Yaskawa INFORM job: DEMO_ROOF_SIDE_0625_3PAINT_11.JBI

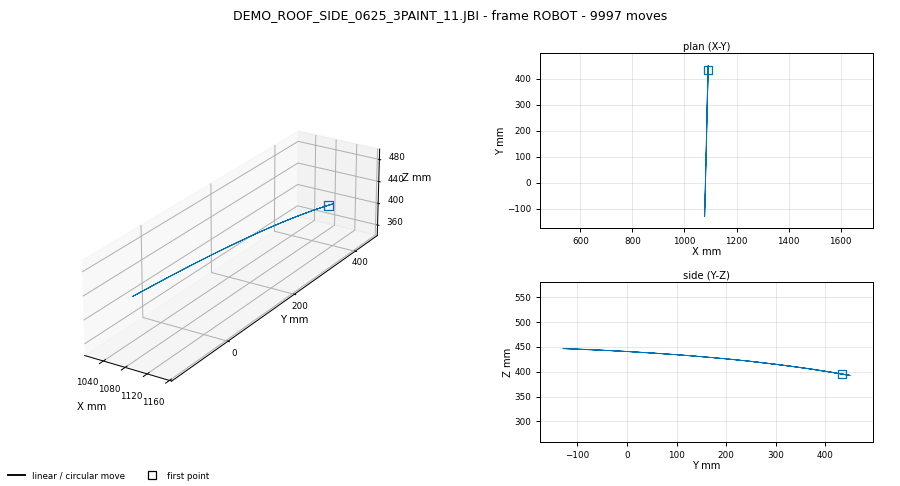
[picture p0: tool path of DEMO_ROOF_SIDE_0625_3PAINT_11.JBI in frame ROBOT, 9997 of 9997 moves have a stored position in this frame; points joined in program order, loops and branches not executed]
/JOB
//NAME DEMO_ROOF_SIDE_0625_3PAINT11
//POS
///NPOS 9997,0,0,0,0,0
///TOOL 0
///USER 0
///POSTYPE ROBOT
///RECTAN
///RCONF 1,0,0,0,0,0,0,0,0,0,0,0,0,0,0,0,0,0,0,0,0,0,0,0
C00000=1091.874,433.807,395.895,178.473,26.068,154.099
C00001=1091.880,434.053,395.852,178.477,26.080,154.102
C00002=1091.887,434.299,395.808,178.480,26.092,154.104
C00003=1091.893,434.545,395.766,178.484,26.104,154.107
C00004=1091.899,434.791,395.723,178.486,26.116,154.110
C00005=1091.906,435.037,395.679,178.490,26.128,154.112
C00006=1091.912,435.283,395.635,178.493,26.141,154.115
C00007=1091.918,435.530,395.592,178.497,26.153,154.117
C00008=1091.926,435.775,395.549,178.500,26.165,154.120
C00009=1091.932,436.022,395.506,178.503,26.177,154.123
C00010=1091.938,436.268,395.462,178.507,26.189,154.126
C00011=1091.945,436.514,395.419,178.510,26.202,154.128
C00012=1091.951,436.760,395.376,178.513,26.214,154.131
C00013=1091.958,437.006,395.332,178.517,26.227,154.134
C00014=1091.965,437.252,395.289,178.520,26.239,154.137
C00015=1091.971,437.498,395.245,178.524,26.252,154.139
C00016=1091.978,437.744,395.201,178.527,26.264,154.142
C00017=1091.988,438.137,395.131,178.533,26.285,154.147
C00018=1091.999,438.531,395.062,178.538,26.305,154.151
C00019=1092.009,438.925,394.992,178.543,26.326,154.156
C00020=1092.020,439.319,394.922,178.548,26.346,154.160
C00021=1092.027,439.565,394.878,178.552,26.359,154.163
C00022=1092.033,439.811,394.834,178.556,26.372,154.166
C00023=1092.041,440.056,394.790,178.559,26.385,154.169
C00024=1092.047,440.302,394.746,178.562,26.398,154.172
C00025=1092.053,440.548,394.703,178.565,26.411,154.175
C00026=1092.060,440.794,394.659,178.569,26.424,154.178
C00027=1092.067,441.041,394.615,178.572,26.438,154.181
C00028=1092.074,441.286,394.570,178.575,26.451,154.184
C00029=1092.080,441.532,394.526,178.579,26.464,154.187
C00030=1092.086,441.778,394.482,178.583,26.478,154.190
C00031=1092.093,442.023,394.438,178.586,26.491,154.193
C00032=1092.100,442.269,394.394,178.589,26.504,154.196
C00033=1092.107,442.516,394.350,178.593,26.518,154.199
C00034=1092.113,442.761,394.305,178.596,26.532,154.202
C00035=1092.120,443.007,394.261,178.600,26.546,154.205
C00036=1092.127,443.253,394.217,178.603,26.559,154.208
C00037=1092.132,443.499,394.172,178.606,26.573,154.211
C00038=1092.140,443.745,394.127,178.610,26.586,154.214
C00039=1092.146,443.991,394.083,178.614,26.601,154.218
C00040=1092.153,444.236,394.039,178.616,26.614,154.221
C00041=1092.159,444.482,393.994,178.620,26.628,154.224
C00042=1092.166,444.728,393.950,178.624,26.642,154.227
C00043=1092.173,444.974,393.906,178.626,26.656,154.230
C00044=1092.180,445.220,393.860,178.629,26.670,154.233
C00045=1092.186,445.466,393.815,178.632,26.684,154.237
C00046=1092.193,445.711,393.772,178.633,26.697,154.240
C00047=1092.200,445.958,393.727,178.636,26.711,154.243
C00048=1092.206,446.203,393.682,178.638,26.725,154.246
C00049=1092.213,446.449,393.637,178.639,26.739,154.250
C00050=1092.220,446.695,393.592,178.641,26.752,154.253
C00051=1092.227,446.940,393.547,178.643,26.767,154.256
C00052=1092.233,447.186,393.502,178.644,26.780,154.260
C00053=1092.240,447.432,393.457,178.645,26.794,154.263
C00054=1092.246,447.677,393.412,178.646,26.807,154.267
C00055=1092.254,447.923,393.367,178.647,26.821,154.270
C00056=1092.260,448.169,393.323,178.648,26.835,154.273
C00057=1092.267,448.415,393.277,178.648,26.849,154.277
C00058=1092.274,448.660,393.233,178.649,26.862,154.280
C00059=1092.281,448.907,393.188,178.649,26.876,154.284
C00060=1092.287,449.152,393.143,178.650,26.890,154.287
C00061=1092.294,449.398,393.098,178.649,26.903,154.291
C00062=1092.301,449.644,393.053,178.649,26.917,154.294
C00063=1092.308,449.888,393.008,178.649,26.931,154.298
C00064=1092.317,450.135,392.964,178.649,26.943,154.301
C00065=1091.932,450.127,392.783,178.601,27.145,154.357
C00066=1091.923,449.881,392.827,178.601,27.132,154.354
C00067=1091.915,449.636,392.873,178.601,27.119,154.350
C00068=1091.908,449.390,392.918,178.601,27.105,154.347
C00069=1091.902,449.145,392.963,178.601,27.091,154.343
C00070=1091.895,448.899,393.008,178.601,27.078,154.340
C00071=1091.888,448.654,393.053,178.601,27.064,154.336
C00072=1091.881,448.407,393.098,178.600,27.050,154.333
C00073=1091.875,448.162,393.143,178.600,27.037,154.330
C00074=1091.868,447.916,393.189,178.599,27.023,154.326
C00075=1091.861,447.670,393.233,178.598,27.009,154.323
C00076=1091.854,447.424,393.278,178.596,26.995,154.319
C00077=1091.848,447.179,393.323,178.595,26.982,154.316
C00078=1091.841,446.933,393.368,178.594,26.968,154.313
C00079=1091.834,446.687,393.413,178.592,26.954,154.309
C00080=1091.827,446.441,393.458,178.591,26.940,154.306
C00081=1091.821,446.196,393.503,178.588,26.926,154.303
C00082=1091.814,445.950,393.547,178.586,26.912,154.299
C00083=1091.807,445.704,393.593,178.585,26.898,154.296
C00084=1091.800,445.458,393.637,178.582,26.884,154.293
C00085=1091.793,445.212,393.682,178.579,26.871,154.290
C00086=1091.787,444.966,393.726,178.576,26.857,154.286
C00087=1091.780,444.721,393.771,178.573,26.843,154.283
C00088=1091.773,444.475,393.816,178.570,26.829,154.280
C00089=1091.767,444.229,393.861,178.567,26.815,154.277
C00090=1091.760,443.983,393.905,178.563,26.801,154.274
C00091=1091.753,443.737,393.950,178.559,26.787,154.270
C00092=1091.746,443.492,393.994,178.556,26.773,154.267
C00093=1091.740,443.246,394.038,178.553,26.760,154.264
C00094=1091.733,443.001,394.083,178.549,26.746,154.261
C00095=1091.727,442.754,394.127,178.545,26.732,154.258
C00096=1091.720,442.508,394.172,178.542,26.718,154.255
C00097=1091.714,442.262,394.216,178.539,26.705,154.252
C00098=1091.707,442.017,394.260,178.535,26.691,154.249
C00099=1091.700,441.770,394.305,178.531,26.678,154.246
C00100=1091.693,441.525,394.349,178.527,26.664,154.243
C00101=1091.687,441.279,394.393,178.525,26.651,154.240
C00102=1091.680,441.033,394.437,178.521,26.637,154.237
C00103=1091.674,440.788,394.481,178.517,26.624,154.234
C00104=1091.667,440.542,394.525,178.514,26.611,154.231
C00105=1091.660,440.296,394.569,178.510,26.598,154.228
C00106=1091.653,440.049,394.613,178.508,26.585,154.225
C00107=1091.646,439.804,394.657,178.504,26.572,154.222
C00108=1091.640,439.558,394.701,178.500,26.559,154.219
C00109=1091.633,439.312,394.745,178.497,26.546,154.216
C00110=1091.622,438.929,394.813,178.491,26.526,154.212
C00111=1091.612,438.547,394.881,178.486,26.506,154.207
C00112=1091.602,438.165,394.950,178.481,26.486,154.203
C00113=1091.592,437.783,395.017,178.475,26.466,154.198
C00114=1091.585,437.537,395.061,178.471,26.454,154.196
C00115=1091.579,437.291,395.104,178.469,26.441,154.193
C00116=1091.572,437.045,395.147,178.465,26.428,154.190
C00117=1091.566,436.799,395.191,178.462,26.416,154.187
C00118=1091.559,436.553,395.235,178.458,26.403,154.185
C00119=1091.552,436.307,395.278,178.455,26.391,154.182
C00120=1091.546,436.061,395.322,178.451,26.378,154.179
C00121=1091.540,435.815,395.365,178.448,26.367,154.176
C00122=1091.532,435.569,395.409,178.444,26.354,154.174
C00123=1091.526,435.322,395.452,178.441,26.342,154.171
C00124=1091.520,435.076,395.496,178.437,26.329,154.168
C00125=1091.513,434.831,395.539,178.434,26.317,154.166
C00126=1091.507,434.584,395.582,178.431,26.305,154.163
C00127=1091.500,434.338,395.626,178.427,26.293,154.160
C00128=1091.493,434.092,395.668,178.424,26.281,154.158
C00129=1091.487,433.846,395.712,178.420,26.268,154.155
C00130=1091.481,433.600,395.754,178.417,26.257,154.152
C00131=1091.474,433.354,395.798,178.414,26.245,154.150
C00132=1091.468,433.108,395.841,178.410,26.233,154.147
C00133=1091.461,432.861,395.884,178.407,26.221,154.144
C00134=1091.455,432.615,395.928,178.403,26.209,154.142
C00135=1091.448,432.369,395.970,178.400,26.197,154.139
C00136=1091.441,432.123,396.013,178.397,26.186,154.137
C00137=1091.436,431.877,396.056,178.393,26.174,154.134
C00138=1091.428,431.631,396.099,178.390,26.162,154.132
C00139=1091.422,431.385,396.142,178.387,26.151,154.129
C00140=1091.415,431.138,396.185,178.383,26.139,154.127
C00141=1091.409,430.892,396.227,178.380,26.128,154.124
C00142=1091.403,430.646,396.270,178.377,26.117,154.122
C00143=1091.396,430.400,396.312,178.374,26.105,154.119
C00144=1091.389,430.154,396.355,178.370,26.094,154.117
C00145=1091.383,429.907,396.398,178.367,26.082,154.114
C00146=1091.377,429.662,396.440,178.364,26.071,154.112
C00147=1091.370,429.415,396.483,178.360,26.060,154.110
C00148=1091.364,429.169,396.526,178.356,26.048,154.107
C00149=1091.358,428.923,396.568,178.353,26.037,154.105
C00150=1091.351,428.677,396.611,178.350,26.026,154.102
C00151=1091.345,428.430,396.654,178.347,26.015,154.100
C00152=1091.338,428.184,396.696,178.343,26.004,154.097
C00153=1091.332,427.938,396.739,178.340,25.993,154.095
C00154=1091.325,427.691,396.780,178.337,25.982,154.093
C00155=1091.318,427.445,396.823,178.333,25.971,154.090
C00156=1091.312,427.200,396.865,178.330,25.960,154.088
C00157=1091.305,426.953,396.908,178.326,25.949,154.086
C00158=1091.299,426.706,396.950,178.323,25.938,154.083
C00159=1091.293,426.460,396.992,178.320,25.927,154.081
C00160=1091.287,426.214,397.034,178.317,25.916,154.079
C00161=1091.280,425.967,397.077,178.313,25.906,154.077
C00162=1091.273,425.736,397.116,178.310,25.895,154.074
C00163=1091.268,425.503,397.156,178.307,25.885,154.072
C00164=1091.261,425.271,397.196,178.304,25.876,154.070
C00165=1091.256,425.039,397.235,178.301,25.866,154.068
C00166=1091.249,424.807,397.275,178.298,25.856,154.066
C00167=1091.244,424.574,397.314,178.294,25.846,154.064
C00168=1091.238,424.343,397.354,178.292,25.836,154.062
C00169=1091.231,424.110,397.393,178.288,25.826,154.060
C00170=1091.225,423.864,397.435,178.285,25.815,154.057
C00171=1091.218,423.618,397.477,178.282,25.805,154.055
C00172=1091.213,423.371,397.519,178.279,25.794,154.053
C00173=1091.206,423.124,397.560,178.275,25.784,154.051
C00174=1091.200,422.879,397.603,178.272,25.774,154.049
C00175=1091.193,422.632,397.644,178.269,25.764,154.046
C00176=1091.187,422.386,397.686,178.266,25.753,154.044
C00177=1091.181,422.139,397.728,178.262,25.743,154.042
C00178=1091.175,421.893,397.769,178.259,25.733,154.040
C00179=1091.168,421.646,397.812,178.256,25.723,154.038
C00180=1091.162,421.400,397.853,178.252,25.713,154.036
C00181=1091.155,421.154,397.894,178.249,25.703,154.034
C00182=1091.149,420.907,397.936,178.246,25.693,154.032
C00183=1091.142,420.660,397.978,178.243,25.682,154.029
C00184=1091.136,420.414,398.019,178.239,25.672,154.027
C00185=1091.130,420.168,398.061,178.236,25.662,154.025
C00186=1091.123,419.921,398.102,178.233,25.653,154.023
C00187=1091.117,419.675,398.143,178.229,25.642,154.021
C00188=1091.110,419.428,398.185,178.226,25.633,154.019
C00189=1091.105,419.182,398.227,178.223,25.623,154.017
C00190=1091.098,418.936,398.267,178.219,25.613,154.015
C00191=1091.092,418.689,398.309,178.217,25.603,154.013
C00192=1091.086,418.442,398.350,178.214,25.594,154.011
C00193=1091.079,418.197,398.391,178.210,25.584,154.009
C00194=1091.072,417.950,398.433,178.207,25.574,154.007
C00195=1091.067,417.703,398.473,178.204,25.564,154.005
C00196=1091.061,417.457,398.515,178.200,25.555,154.003
C00197=1091.054,417.210,398.556,178.197,25.545,154.001
C00198=1091.048,416.963,398.597,178.194,25.536,153.999
C00199=1091.042,416.717,398.638,178.191,25.526,153.997
C00200=1091.035,416.471,398.679,178.187,25.517,153.995
C00201=1091.029,416.224,398.720,178.184,25.507,153.993
C00202=1091.022,415.978,398.761,178.181,25.497,153.991
C00203=1091.017,415.731,398.802,178.177,25.488,153.989
C00204=1091.009,415.484,398.843,178.175,25.479,153.987
C00205=1091.004,415.237,398.884,178.171,25.470,153.985
C00206=1090.997,414.992,398.925,178.168,25.461,153.984
C00207=1090.991,414.744,398.966,178.165,25.451,153.982
C00208=1090.984,414.498,399.006,178.162,25.442,153.980
C00209=1090.978,414.252,399.047,178.159,25.433,153.978
C00210=1090.972,414.005,399.088,178.155,25.424,153.976
C00211=1090.965,413.759,399.128,178.152,25.414,153.974
C00212=1090.959,413.511,399.170,178.149,25.405,153.972
C00213=1090.953,413.265,399.210,178.146,25.396,153.970
C00214=1090.946,413.018,399.250,178.142,25.387,153.969
C00215=1090.940,412.772,399.291,178.140,25.378,153.967
C00216=1090.934,412.526,399.331,178.136,25.369,153.965
C00217=1090.928,412.278,399.373,178.133,25.360,153.963
C00218=1090.922,412.054,399.409,178.130,25.352,153.961
C00219=1090.917,411.829,399.446,178.127,25.344,153.960
C00220=1090.911,411.605,399.483,178.124,25.336,153.958
C00221=1090.905,411.380,399.520,178.122,25.328,153.957
C00222=1090.899,411.155,399.557,178.119,25.319,153.955
C00223=1090.894,410.930,399.594,178.115,25.311,153.953
C00224=1090.887,410.706,399.630,178.112,25.303,153.952
C00225=1090.882,410.481,399.667,178.110,25.295,153.950
C00226=1090.876,410.234,399.707,178.107,25.287,153.948
C00227=1090.870,409.987,399.748,178.103,25.278,153.947
C00228=1090.864,409.741,399.788,178.100,25.269,153.945
C00229=1090.857,409.494,399.829,178.097,25.260,153.943
C00230=1090.852,409.247,399.869,178.094,25.252,153.941
C00231=1090.845,409.001,399.909,178.091,25.243,153.939
C00232=1090.839,408.754,399.949,178.088,25.234,153.938
C00233=1090.833,408.507,399.989,178.084,25.226,153.936
C00234=1090.827,408.260,400.030,178.082,25.217,153.934
C00235=1090.821,408.014,400.070,178.078,25.208,153.933
C00236=1090.814,407.767,400.110,178.075,25.200,153.931
C00237=1090.808,407.520,400.149,178.072,25.192,153.929
C00238=1090.802,407.274,400.190,178.069,25.183,153.927
C00239=1090.795,407.027,400.230,178.065,25.175,153.926
C00240=1090.790,406.780,400.271,178.063,25.166,153.924
C00241=1090.784,406.533,400.310,178.059,25.158,153.923
C00242=1090.777,406.287,400.350,178.057,25.149,153.921
C00243=1090.772,406.041,400.390,178.053,25.141,153.919
C00244=1090.766,405.794,400.429,178.050,25.133,153.918
C00245=1090.759,405.547,400.469,178.047,25.124,153.916
C00246=1090.753,405.300,400.509,178.044,25.116,153.914
C00247=1090.747,405.054,400.549,178.040,25.108,153.913
C00248=1090.741,404.806,400.588,178.038,25.100,153.911
C00249=1090.734,404.560,400.629,178.035,25.092,153.909
C00250=1090.728,404.313,400.668,178.031,25.084,153.908
C00251=1090.722,404.066,400.708,178.029,25.076,153.906
C00252=1090.716,403.819,400.748,178.025,25.067,153.905
C00253=1090.710,403.573,400.787,178.022,25.059,153.903
C00254=1090.703,403.326,400.826,178.018,25.051,153.902
C00255=1090.697,403.079,400.866,178.016,25.043,153.900
C00256=1090.691,402.833,400.906,178.013,25.035,153.898
C00257=1090.685,402.586,400.945,178.009,25.027,153.897
C00258=1090.679,402.339,400.985,178.007,25.019,153.895
C00259=1090.672,402.091,401.024,178.004,25.011,153.894
C00260=1090.667,401.846,401.064,178.000,25.003,153.892
C00261=1090.660,401.599,401.103,177.997,24.996,153.891
C00262=1090.654,401.352,401.142,177.994,24.988,153.889
C00263=1090.648,401.105,401.182,177.991,24.980,153.888
C00264=1090.642,400.859,401.221,177.988,24.972,153.886
C00265=1090.636,400.612,401.261,177.984,24.964,153.885
C00266=1090.629,400.365,401.300,177.982,24.956,153.883
C00267=1090.623,400.118,401.339,177.979,24.949,153.882
C00268=1090.617,399.871,401.378,177.975,24.941,153.880
C00269=1090.611,399.624,401.418,177.972,24.933,153.878
C00270=1090.605,399.377,401.457,177.970,24.925,153.877
C00271=1090.599,399.130,401.496,177.967,24.918,153.876
C00272=1090.593,398.884,401.535,177.963,24.910,153.874
C00273=1090.586,398.637,401.574,177.960,24.903,153.873
C00274=1090.581,398.413,401.610,177.957,24.896,153.871
C00275=1090.575,398.188,401.645,177.954,24.889,153.870
C00276=1090.570,397.964,401.680,177.952,24.882,153.869
C00277=1090.564,397.740,401.717,177.949,24.875,153.867
C00278=1090.558,397.515,401.751,177.946,24.868,153.866
C00279=1090.553,397.291,401.787,177.943,24.862,153.865
C00280=1090.547,397.067,401.823,177.941,24.855,153.863
C00281=1090.543,396.843,401.858,177.938,24.848,153.862
C00282=1090.536,396.596,401.897,177.935,24.841,153.861
C00283=1090.530,396.349,401.936,177.931,24.833,153.859
C00284=1090.524,396.102,401.974,177.929,24.826,153.858
C00285=1090.518,395.855,402.013,177.926,24.818,153.857
C00286=1090.512,395.609,402.052,177.923,24.811,153.855
C00287=1090.506,395.361,402.090,177.919,24.803,153.854
C00288=1090.500,395.114,402.130,177.916,24.796,153.852
C00289=1090.493,394.868,402.168,177.913,24.789,153.851
C00290=1090.487,394.621,402.207,177.910,24.782,153.850
C00291=1090.481,394.374,402.245,177.907,24.774,153.848
C00292=1090.475,394.127,402.284,177.904,24.767,153.847
C00293=1090.469,393.880,402.323,177.901,24.760,153.846
C00294=1090.463,393.633,402.361,177.898,24.753,153.844
C00295=1090.457,393.387,402.399,177.895,24.746,153.843
C00296=1090.451,393.140,402.439,177.892,24.738,153.841
C00297=1090.444,392.893,402.477,177.889,24.731,153.840
C00298=1090.439,392.646,402.516,177.885,24.724,153.839
C00299=1090.433,392.400,402.554,177.882,24.717,153.838
C00300=1090.426,392.152,402.592,177.879,24.710,153.836
C00301=1090.421,391.905,402.631,177.876,24.703,153.835
C00302=1090.414,391.658,402.670,177.873,24.696,153.834
C00303=1090.408,391.412,402.707,177.870,24.689,153.832
C00304=1090.401,391.165,402.746,177.866,24.682,153.831
C00305=1090.395,390.918,402.784,177.864,24.675,153.830
C00306=1090.390,390.670,402.823,177.860,24.668,153.829
C00307=1090.383,390.424,402.861,177.858,24.661,153.827
C00308=1090.378,390.177,402.899,177.855,24.654,153.826
C00309=1090.371,389.930,402.937,177.852,24.648,153.825
C00310=1090.365,389.684,402.975,177.849,24.641,153.823
C00311=1090.358,389.436,403.014,177.846,24.634,153.822
C00312=1090.352,389.190,403.051,177.842,24.627,153.821
C00313=1090.347,388.943,403.090,177.839,24.620,153.820
C00314=1090.341,388.695,403.128,177.836,24.613,153.819
C00315=1090.335,388.449,403.166,177.833,24.606,153.817
C00316=1090.328,388.202,403.204,177.830,24.600,153.816
C00317=1090.322,387.955,403.242,177.827,24.593,153.815
C00318=1090.316,387.708,403.280,177.824,24.586,153.813
C00319=1090.310,387.461,403.318,177.821,24.580,153.812
C00320=1090.304,387.214,403.356,177.818,24.573,153.811
C00321=1090.298,386.967,403.394,177.815,24.566,153.810
C00322=1090.292,386.720,403.431,177.812,24.559,153.809
C00323=1090.285,386.473,403.469,177.807,24.553,153.808
C00324=1090.280,386.226,403.508,177.804,24.546,153.806
C00325=1090.274,385.979,403.546,177.801,24.539,153.805
C00326=1090.268,385.732,403.583,177.798,24.533,153.804
C00327=1090.262,385.485,403.621,177.795,24.526,153.803
C00328=1090.256,385.238,403.659,177.792,24.520,153.802
C00329=1090.250,384.991,403.697,177.789,24.513,153.800
C00330=1090.245,384.774,403.730,177.787,24.507,153.799
C00331=1090.239,384.556,403.764,177.784,24.502,153.798
C00332=1090.235,384.338,403.797,177.781,24.496,153.797
C00333=1090.229,384.121,403.829,177.779,24.490,153.796
C00334=1090.224,383.903,403.863,177.776,24.485,153.795
C00335=1090.218,383.686,403.896,177.774,24.479,153.794
C00336=1090.213,383.468,403.930,177.770,24.473,153.793
C00337=1090.208,383.250,403.962,177.768,24.467,153.792
C00338=1090.202,383.003,404.000,177.765,24.461,153.791
C00339=1090.196,382.757,404.037,177.762,24.454,153.790
C00340=1090.190,382.510,404.075,177.759,24.448,153.789
C00341=1090.184,382.263,404.112,177.756,24.442,153.788
C00342=1090.178,382.015,404.150,177.752,24.435,153.786
C00343=1090.171,381.769,404.188,177.749,24.429,153.785
C00344=1090.166,381.521,404.225,177.746,24.423,153.784
C00345=1090.160,381.275,404.262,177.743,24.416,153.783
C00346=1090.154,381.027,404.299,177.740,24.410,153.782
C00347=1090.147,380.780,404.337,177.737,24.404,153.781
C00348=1090.141,380.533,404.374,177.734,24.397,153.780
C00349=1090.135,380.286,404.412,177.731,24.391,153.779
C00350=1090.130,380.039,404.449,177.727,24.385,153.778
C00351=1090.123,379.792,404.486,177.724,24.379,153.777
C00352=1090.118,379.545,404.523,177.721,24.373,153.776
C00353=1090.112,379.298,404.561,177.718,24.367,153.774
C00354=1090.105,379.051,404.597,177.716,24.361,153.773
C00355=1090.099,378.804,404.635,177.713,24.355,153.772
C00356=1090.093,378.556,404.672,177.709,24.348,153.771
C00357=1090.087,378.309,404.709,177.706,24.342,153.770
C00358=1090.081,378.062,404.746,177.703,24.336,153.769
C00359=1090.075,377.815,404.784,177.700,24.330,153.768
C00360=1090.069,377.568,404.820,177.697,24.324,153.767
C00361=1090.063,377.321,404.858,177.694,24.318,153.766
C00362=1090.058,377.074,404.895,177.690,24.312,153.765
C00363=1090.051,376.827,404.931,177.687,24.306,153.764
C00364=1090.046,376.579,404.968,177.684,24.300,153.763
C00365=1090.040,376.332,405.005,177.682,24.294,153.762
C00366=1090.033,376.086,405.042,177.679,24.288,153.761
C00367=1090.028,375.838,405.079,177.675,24.282,153.760
C00368=1090.021,375.591,405.116,177.672,24.276,153.759
C00369=1090.016,375.344,405.153,177.669,24.270,153.758
C00370=1090.010,375.097,405.190,177.666,24.264,153.757
C00371=1090.004,374.849,405.226,177.663,24.258,153.756
C00372=1089.998,374.602,405.263,177.660,24.252,153.755
C00373=1089.993,374.356,405.300,177.657,24.246,153.754
C00374=1089.987,374.108,405.337,177.654,24.240,153.753
C00375=1089.981,373.861,405.373,177.651,24.235,153.752
C00376=1089.975,373.614,405.410,177.647,24.229,153.751
C00377=1089.969,373.367,405.447,177.644,24.223,153.750
C00378=1089.962,373.120,405.483,177.641,24.217,153.749
C00379=1089.957,372.873,405.520,177.639,24.212,153.748
C00380=1089.950,372.625,405.556,177.635,24.206,153.747
C00381=1089.945,372.378,405.594,177.632,24.200,153.746
C00382=1089.938,372.131,405.630,177.629,24.194,153.745
C00383=1089.932,371.884,405.666,177.626,24.188,153.744
C00384=1089.927,371.637,405.703,177.623,24.183,153.743
C00385=1089.920,371.389,405.739,177.620,24.177,153.742
C00386=1089.910,370.982,405.800,177.615,24.168,153.741
C00387=1089.900,370.574,405.859,177.610,24.158,153.739
C00388=1089.891,370.167,405.919,177.605,24.149,153.738
C00389=1089.881,369.759,405.979,177.599,24.140,153.736
C00390=1089.875,369.511,406.016,177.596,24.134,153.735
C00391=1089.869,369.265,406.052,177.594,24.129,153.734
C00392=1089.863,369.017,406.088,177.590,24.123,153.733
C00393=1089.857,368.770,406.124,177.587,24.118,153.732
C00394=1089.851,368.523,406.161,177.584,24.112,153.731
C00395=1089.845,368.275,406.197,177.580,24.106,153.731
C00396=1089.840,368.029,406.233,177.578,24.101,153.730
C00397=1089.834,367.781,406.269,177.575,24.095,153.729
C00398=1089.828,367.534,406.306,177.571,24.090,153.728
C00399=1089.822,367.286,406.342,177.568,24.084,153.727
C00400=1089.816,367.039,406.378,177.566,24.079,153.726
C00401=1089.810,366.792,406.414,177.563,24.073,153.725
C00402=1089.804,366.545,406.450,177.559,24.068,153.724
C00403=1089.799,366.297,406.486,177.556,24.062,153.723
C00404=1089.793,366.051,406.522,177.553,24.057,153.722
C00405=1089.787,365.803,406.558,177.550,24.052,153.722
C00406=1089.781,365.556,406.594,177.547,24.046,153.721
C00407=1089.774,365.308,406.630,177.544,24.041,153.720
C00408=1089.768,365.061,406.666,177.541,24.035,153.719
C00409=1089.763,364.814,406.701,177.538,24.030,153.718
C00410=1089.757,364.567,406.738,177.534,24.025,153.717
C00411=1089.751,364.319,406.774,177.532,24.019,153.716
C00412=1089.745,364.072,406.809,177.529,24.014,153.716
C00413=1089.739,363.824,406.845,177.525,24.008,153.715
C00414=1089.733,363.577,406.881,177.523,24.003,153.714
C00415=1089.727,363.330,406.917,177.519,23.998,153.713
C00416=1089.721,363.083,406.952,177.516,23.993,153.712
C00417=1089.715,362.835,406.988,177.513,23.987,153.711
C00418=1089.709,362.587,407.024,177.510,23.982,153.711
C00419=1089.704,362.341,407.060,177.507,23.977,153.710
C00420=1089.698,362.093,407.095,177.503,23.971,153.709
C00421=1089.692,361.846,407.131,177.501,23.967,153.708
C00422=1089.686,361.599,407.167,177.498,23.961,153.707
C00423=1089.680,361.351,407.202,177.494,23.956,153.706
C00424=1089.674,361.103,407.238,177.492,23.951,153.706
C00425=1089.669,360.856,407.273,177.488,23.946,153.705
C00426=1089.661,360.572,407.314,177.485,23.940,153.704
C00427=1089.655,360.288,407.355,177.481,23.934,153.703
C00428=1089.648,360.003,407.396,177.478,23.928,153.702
C00429=1089.641,359.719,407.436,177.474,23.922,153.701
C00430=1089.635,359.471,407.472,177.471,23.917,153.700
C00431=1089.630,359.224,407.507,177.468,23.912,153.700
C00432=1089.623,358.977,407.543,177.465,23.907,153.699
C00433=1089.617,358.729,407.578,177.462,23.902,153.698
C00434=1089.612,358.482,407.614,177.458,23.897,153.697
C00435=1089.606,358.234,407.649,177.456,23.892,153.697
C00436=1089.600,357.987,407.683,177.453,23.886,153.696
C00437=1089.594,357.739,407.719,177.450,23.882,153.695
C00438=1089.585,357.384,407.770,177.445,23.875,153.694
C00439=1089.577,357.029,407.821,177.440,23.867,153.693
C00440=1089.568,356.674,407.871,177.437,23.860,153.692
C00441=1089.560,356.319,407.922,177.432,23.853,153.691
C00442=1089.553,356.072,407.957,177.428,23.848,153.690
C00443=1089.548,355.825,407.992,177.426,23.843,153.689
C00444=1089.542,355.577,408.027,177.422,23.838,153.688
C00445=1089.536,355.330,408.062,177.420,23.833,153.688
C00446=1089.530,355.082,408.097,177.416,23.828,153.687
C00447=1089.525,354.835,408.132,177.413,23.823,153.686
C00448=1089.519,354.588,408.167,177.410,23.818,153.685
C00449=1089.513,354.340,408.202,177.407,23.813,153.685
C00450=1089.508,354.093,408.237,177.404,23.809,153.684
C00451=1089.501,353.845,408.272,177.401,23.804,153.683
C00452=1089.496,353.598,408.307,177.398,23.799,153.682
C00453=1089.489,353.350,408.342,177.395,23.794,153.682
C00454=1089.484,353.103,408.377,177.391,23.789,153.681
C00455=1089.478,352.854,408.412,177.389,23.784,153.680
C00456=1089.472,352.608,408.447,177.385,23.779,153.680
C00457=1089.466,352.360,408.482,177.383,23.775,153.679
C00458=1089.460,352.112,408.516,177.379,23.770,153.678
C00459=1089.454,351.865,408.551,177.377,23.765,153.678
C00460=1089.448,351.617,408.586,177.373,23.761,153.677
C00461=1089.442,351.371,408.620,177.371,23.756,153.676
C00462=1089.437,351.122,408.655,177.367,23.751,153.676
C00463=1089.431,350.875,408.689,177.364,23.746,153.675
C00464=1089.425,350.627,408.724,177.361,23.742,153.674
C00465=1089.419,350.380,408.759,177.357,23.737,153.673
C00466=1089.414,350.132,408.794,177.355,23.732,153.673
C00467=1089.407,349.885,408.828,177.351,23.727,153.672
C00468=1089.401,349.638,408.863,177.349,23.723,153.671
C00469=1089.395,349.390,408.898,177.345,23.718,153.671
C00470=1089.390,349.142,408.932,177.343,23.714,153.670
C00471=1089.384,348.895,408.967,177.339,23.709,153.669
C00472=1089.378,348.647,409.001,177.337,23.704,153.669
C00473=1089.372,348.399,409.035,177.333,23.699,153.668
C00474=1089.367,348.152,409.070,177.330,23.695,153.667
C00475=1089.360,347.904,409.105,177.327,23.690,153.667
C00476=1089.354,347.657,409.139,177.324,23.685,153.666
C00477=1089.349,347.410,409.174,177.321,23.681,153.665
C00478=1089.343,347.162,409.208,177.318,23.676,153.665
C00479=1089.337,346.914,409.242,177.315,23.671,153.664
C00480=1089.332,346.667,409.277,177.312,23.667,153.663
C00481=1089.326,346.419,409.311,177.308,23.662,153.663
C00482=1089.319,346.171,409.345,177.306,23.658,153.662
C00483=1089.314,345.924,409.380,177.302,23.653,153.661
C00484=1089.308,345.677,409.414,177.300,23.649,153.661
C00485=1089.302,345.429,409.448,177.296,23.644,153.660
C00486=1089.296,345.181,409.482,177.293,23.639,153.659
C00487=1089.291,344.934,409.517,177.290,23.635,153.659
C00488=1089.285,344.686,409.550,177.287,23.630,153.658
C00489=1089.279,344.438,409.585,177.284,23.626,153.658
C00490=1089.270,344.049,409.638,177.279,23.619,153.657
C00491=1089.261,343.660,409.692,177.274,23.612,153.656
C00492=1089.251,343.270,409.746,177.269,23.605,153.655
C00493=1089.242,342.881,409.799,177.265,23.598,153.654
C00494=1089.236,342.633,409.833,177.262,23.594,153.653
C00495=1089.231,342.386,409.867,177.259,23.589,153.652
C00496=1089.225,342.138,409.901,177.255,23.585,153.652
C00497=1089.218,341.890,409.935,177.253,23.581,153.651
C00498=1089.213,341.643,409.969,177.249,23.576,153.651
C00499=1089.207,341.395,410.003,177.246,23.571,153.650
C00500=1089.201,341.148,410.037,177.243,23.567,153.650
C00501=1089.195,340.900,410.070,177.240,23.563,153.649
C00502=1089.189,340.652,410.105,177.237,23.558,153.648
C00503=1089.183,340.404,410.138,177.234,23.554,153.648
C00504=1089.178,340.157,410.172,177.231,23.550,153.647
C00505=1089.172,339.909,410.205,177.228,23.545,153.647
C00506=1089.166,339.662,410.239,177.225,23.541,153.646
C00507=1089.160,339.414,410.273,177.222,23.537,153.645
C00508=1089.155,339.166,410.307,177.219,23.532,153.645
C00509=1089.149,338.919,410.341,177.216,23.528,153.644
C00510=1089.143,338.671,410.374,177.212,23.523,153.644
C00511=1089.137,338.423,410.408,177.210,23.519,153.643
C00512=1089.131,338.175,410.442,177.207,23.515,153.643
C00513=1089.126,337.927,410.475,177.203,23.511,153.642
C00514=1089.120,337.680,410.509,177.200,23.507,153.641
C00515=1089.114,337.432,410.543,177.198,23.503,153.641
C00516=1089.108,337.185,410.577,177.194,23.498,153.640
C00517=1089.102,336.937,410.609,177.191,23.494,153.640
C00518=1089.097,336.690,410.643,177.188,23.489,153.639
C00519=1089.091,336.442,410.677,177.185,23.485,153.639
C00520=1089.085,336.194,410.710,177.182,23.481,153.638
C00521=1089.079,335.946,410.744,177.179,23.477,153.637
C00522=1089.073,335.698,410.777,177.176,23.473,153.637
C00523=1089.067,335.451,410.811,177.173,23.468,153.636
C00524=1089.061,335.203,410.844,177.170,23.464,153.636
C00525=1089.056,334.955,410.877,177.167,23.460,153.635
C00526=1089.050,334.707,410.911,177.164,23.456,153.635
C00527=1089.044,334.460,410.944,177.160,23.452,153.634
C00528=1089.038,334.212,410.977,177.158,23.448,153.634
C00529=1089.033,333.964,411.011,177.155,23.444,153.633
C00530=1089.027,333.716,411.044,177.151,23.439,153.633
C00531=1089.021,333.469,411.077,177.149,23.435,153.632
C00532=1089.015,333.221,411.110,177.146,23.431,153.631
C00533=1089.010,332.973,411.144,177.142,23.427,153.631
C00534=1089.004,332.725,411.177,177.139,23.423,153.630
C00535=1088.997,332.478,411.210,177.137,23.419,153.630
C00536=1088.992,332.230,411.244,177.133,23.414,153.629
C00537=1088.986,331.982,411.277,177.130,23.410,153.629
C00538=1088.980,331.735,411.310,177.128,23.406,153.628
C00539=1088.974,331.487,411.343,177.124,23.402,153.628
C00540=1088.968,331.239,411.376,177.121,23.398,153.627
C00541=1088.963,330.991,411.409,177.118,23.394,153.627
C00542=1088.953,330.596,411.461,177.113,23.388,153.626
C00543=1088.944,330.201,411.514,177.108,23.382,153.625
C00544=1088.935,329.806,411.566,177.103,23.375,153.624
C00545=1088.925,329.411,411.619,177.098,23.369,153.624
C00546=1088.919,329.164,411.652,177.095,23.365,153.623
C00547=1088.914,328.915,411.684,177.092,23.361,153.623
C00548=1088.907,328.667,411.717,177.090,23.357,153.622
C00549=1088.901,328.420,411.750,177.086,23.353,153.622
C00550=1088.896,328.172,411.783,177.083,23.349,153.621
C00551=1088.889,327.924,411.816,177.080,23.345,153.621
C00552=1088.884,327.676,411.848,177.077,23.341,153.620
C00553=1088.878,327.428,411.881,177.074,23.337,153.620
C00554=1088.871,327.181,411.914,177.071,23.334,153.619
C00555=1088.867,326.933,411.946,177.068,23.329,153.619
C00556=1088.860,326.685,411.979,177.065,23.325,153.618
C00557=1088.854,326.438,412.012,177.062,23.322,153.618
C00558=1088.849,326.189,412.044,177.059,23.318,153.617
C00559=1088.843,325.942,412.077,177.056,23.314,153.617
C00560=1088.837,325.694,412.110,177.052,23.310,153.617
C00561=1088.831,325.445,412.142,177.050,23.306,153.616
C00562=1088.825,325.199,412.175,177.047,23.302,153.616
C00563=1088.819,324.951,412.207,177.044,23.299,153.615
C00564=1088.814,324.702,412.240,177.040,23.294,153.615
C00565=1088.808,324.455,412.273,177.037,23.290,153.614
C00566=1088.802,324.207,412.305,177.035,23.287,153.614
C00567=1088.797,323.959,412.338,177.032,23.283,153.613
C00568=1088.791,323.711,412.370,177.029,23.279,153.613
C00569=1088.784,323.464,412.403,177.025,23.275,153.612
C00570=1088.779,323.215,412.435,177.022,23.271,153.612
C00571=1088.773,322.968,412.468,177.020,23.268,153.611
C00572=1088.767,322.720,412.500,177.017,23.264,153.611
C00573=1088.761,322.472,412.532,177.014,23.260,153.610
C00574=1088.756,322.225,412.565,177.010,23.256,153.610
C00575=1088.750,321.976,412.597,177.007,23.252,153.610
C00576=1088.744,321.729,412.629,177.004,23.248,153.609
C00577=1088.738,321.481,412.661,177.002,23.245,153.609
C00578=1088.734,321.233,412.694,176.998,23.240,153.608
C00579=1088.727,320.985,412.726,176.995,23.237,153.608
C00580=1088.721,320.737,412.758,176.992,23.233,153.607
C00581=1088.716,320.489,412.790,176.989,23.229,153.607
C00582=1088.710,320.241,412.823,176.987,23.226,153.606
C00583=1088.704,319.993,412.855,176.984,23.222,153.606
C00584=1088.699,319.746,412.887,176.980,23.217,153.605
C00585=1088.693,319.498,412.919,176.977,23.214,153.605
C00586=1088.687,319.251,412.952,176.974,23.210,153.605
C00587=1088.682,319.002,412.984,176.972,23.206,153.604
C00588=1088.676,318.754,413.016,176.969,23.203,153.604
C00589=1088.671,318.506,413.048,176.965,23.199,153.603
C00590=1088.665,318.258,413.080,176.962,23.195,153.603
C00591=1088.659,318.011,413.112,176.959,23.191,153.602
C00592=1088.653,317.763,413.144,176.956,23.188,153.602
C00593=1088.648,317.515,413.177,176.954,23.184,153.602
C00594=1088.639,317.113,413.229,176.949,23.178,153.601
C00595=1088.630,316.711,413.280,176.944,23.171,153.600
C00596=1088.621,316.309,413.332,176.939,23.166,153.599
C00597=1088.612,315.907,413.384,176.934,23.159,153.599
C00598=1088.606,315.659,413.415,176.931,23.156,153.598
C00599=1088.600,315.411,413.447,176.929,23.152,153.598
C00600=1088.595,315.163,413.479,176.925,23.148,153.597
C00601=1088.589,314.915,413.511,176.922,23.144,153.597
C00602=1088.583,314.667,413.543,176.919,23.141,153.597
C00603=1088.577,314.420,413.574,176.916,23.138,153.596
C00604=1088.571,314.171,413.606,176.913,23.134,153.596
C00605=1088.565,313.924,413.638,176.910,23.131,153.595
C00606=1088.559,313.676,413.670,176.907,23.127,153.595
C00607=1088.553,313.428,413.701,176.904,23.123,153.595
C00608=1088.547,313.180,413.733,176.901,23.120,153.594
C00609=1088.541,312.932,413.765,176.898,23.116,153.594
C00610=1088.536,312.684,413.796,176.895,23.112,153.593
C00611=1088.530,312.436,413.827,176.892,23.109,153.593
C00612=1088.524,312.189,413.859,176.889,23.106,153.593
C00613=1088.518,311.940,413.891,176.886,23.102,153.592
C00614=1088.512,311.693,413.922,176.883,23.099,153.592
C00615=1088.506,311.444,413.953,176.879,23.095,153.592
C00616=1088.501,311.197,413.985,176.876,23.091,153.591
C00617=1088.494,310.949,414.017,176.873,23.088,153.591
C00618=1088.489,310.701,414.048,176.871,23.084,153.590
C00619=1088.483,310.453,414.079,176.868,23.081,153.590
C00620=1088.478,310.205,414.111,176.865,23.077,153.590
C00621=1088.471,309.957,414.143,176.862,23.074,153.589
C00622=1088.466,309.709,414.174,176.859,23.070,153.589
C00623=1088.459,309.461,414.205,176.856,23.067,153.589
C00624=1088.454,309.213,414.236,176.853,23.064,153.588
C00625=1088.449,308.965,414.268,176.849,23.059,153.588
C00626=1088.442,308.718,414.299,176.846,23.056,153.588
C00627=1088.437,308.469,414.330,176.843,23.053,153.587
C00628=1088.431,308.221,414.362,176.841,23.049,153.587
C00629=1088.425,307.973,414.392,176.838,23.046,153.586
C00630=1088.420,307.726,414.424,176.835,23.042,153.586
C00631=1088.413,307.477,414.455,176.832,23.039,153.586
C00632=1088.408,307.230,414.486,176.829,23.035,153.585
C00633=1088.403,306.982,414.517,176.826,23.032,153.585
C00634=1088.396,306.734,414.549,176.823,23.028,153.584
C00635=1088.391,306.486,414.580,176.820,23.025,153.584
C00636=1088.385,306.238,414.611,176.816,23.021,153.584
C00637=1088.379,305.990,414.642,176.813,23.018,153.583
C00638=1088.373,305.742,414.673,176.810,23.014,153.583
C00639=1088.368,305.494,414.704,176.807,23.011,153.583
C00640=1088.361,305.246,414.736,176.805,23.007,153.582
C00641=1088.356,304.998,414.766,176.802,23.004,153.582
C00642=1088.351,304.750,414.797,176.799,23.000,153.582
C00643=1088.345,304.503,414.828,176.796,22.997,153.581
C00644=1088.339,304.254,414.860,176.793,22.994,153.581
C00645=1088.334,304.006,414.890,176.790,22.990,153.581
C00646=1088.324,303.607,414.940,176.785,22.984,153.580
C00647=1088.315,303.208,414.990,176.780,22.979,153.579
C00648=1088.306,302.808,415.040,176.775,22.973,153.579
C00649=1088.298,302.410,415.090,176.771,22.968,153.578
C00650=1088.291,302.161,415.120,176.768,22.965,153.578
C00651=1088.286,301.913,415.151,176.765,22.961,153.577
C00652=1088.280,301.665,415.182,176.762,22.958,153.577
C00653=1088.275,301.418,415.213,176.759,22.954,153.577
C00654=1088.269,301.170,415.244,176.755,22.950,153.576
C00655=1088.264,300.922,415.274,176.752,22.947,153.576
C00656=1088.257,300.673,415.305,176.749,22.944,153.576
C00657=1088.252,300.426,415.336,176.746,22.940,153.575
C00658=1088.247,300.177,415.366,176.744,22.937,153.575
C00659=1088.241,299.930,415.397,176.741,22.934,153.575
C00660=1088.236,299.681,415.428,176.738,22.930,153.574
C00661=1088.230,299.434,415.458,176.735,22.927,153.574
C00662=1088.225,299.185,415.489,176.732,22.923,153.574
C00663=1088.219,298.938,415.519,176.729,22.920,153.573
C00664=1088.213,298.689,415.550,176.726,22.917,153.573
C00665=1088.207,298.441,415.581,176.723,22.913,153.573
C00666=1088.202,298.193,415.611,176.720,22.910,153.572
C00667=1088.196,297.945,415.642,176.717,22.906,153.572
C00668=1088.191,297.697,415.673,176.714,22.903,153.572
C00669=1088.185,297.449,415.703,176.711,22.900,153.571
C00670=1088.179,297.202,415.733,176.708,22.896,153.571
C00671=1088.173,296.954,415.764,176.705,22.893,153.571
C00672=1088.167,296.705,415.795,176.702,22.889,153.570
C00673=1088.162,296.456,415.825,176.699,22.886,153.570
C00674=1088.156,296.209,415.855,176.696,22.883,153.570
C00675=1088.150,295.961,415.885,176.693,22.880,153.569
C00676=1088.145,295.713,415.916,176.690,22.877,153.569
C00677=1088.139,295.465,415.946,176.687,22.873,153.569
C00678=1088.133,295.217,415.977,176.684,22.870,153.568
C00679=1088.128,294.969,416.006,176.681,22.866,153.568
C00680=1088.122,294.721,416.036,176.678,22.863,153.568
C00681=1088.116,294.473,416.067,176.675,22.860,153.568
C00682=1088.110,294.224,416.098,176.672,22.857,153.567
C00683=1088.105,293.976,416.128,176.669,22.854,153.567
C00684=1088.099,293.728,416.158,176.666,22.850,153.567
C00685=1088.093,293.480,416.188,176.664,22.847,153.566
C00686=1088.088,293.232,416.218,176.661,22.844,153.566
C00687=1088.082,292.984,416.248,176.659,22.841,153.566
C00688=1088.076,292.736,416.279,176.656,22.838,153.565
C00689=1088.070,292.488,416.308,176.653,22.834,153.565
C00690=1088.065,292.240,416.339,176.650,22.831,153.565
C00691=1088.059,291.992,416.368,176.647,22.828,153.564
C00692=1088.053,291.744,416.399,176.644,22.825,153.564
C00693=1088.047,291.496,416.429,176.641,22.821,153.564
C00694=1088.042,291.247,416.459,176.638,22.818,153.564
C00695=1088.036,291.000,416.489,176.635,22.815,153.563
C00696=1088.031,290.751,416.519,176.632,22.812,153.563
C00697=1088.025,290.503,416.549,176.629,22.808,153.563
C00698=1088.016,290.119,416.595,176.624,22.804,153.562
C00699=1088.007,289.733,416.641,176.620,22.799,153.562
C00700=1087.999,289.348,416.688,176.615,22.793,153.561
C00701=1087.989,288.962,416.734,176.611,22.789,153.561
C00702=1087.983,288.714,416.764,176.608,22.786,153.561
C00703=1087.978,288.466,416.794,176.605,22.782,153.560
C00704=1087.972,288.218,416.824,176.602,22.779,153.560
C00705=1087.966,287.970,416.853,176.599,22.776,153.560
C00706=1087.960,287.722,416.883,176.596,22.773,153.559
C00707=1087.954,287.474,416.913,176.593,22.770,153.559
C00708=1087.949,287.225,416.943,176.590,22.766,153.559
C00709=1087.944,286.978,416.972,176.587,22.763,153.558
C00710=1087.937,286.730,417.002,176.584,22.760,153.558
C00711=1087.932,286.482,417.031,176.581,22.757,153.558
C00712=1087.926,286.233,417.061,176.578,22.753,153.558
C00713=1087.921,285.985,417.091,176.575,22.751,153.557
C00714=1087.915,285.737,417.120,176.572,22.748,153.557
C00715=1087.909,285.489,417.150,176.570,22.745,153.557
C00716=1087.903,285.240,417.180,176.567,22.741,153.557
C00717=1087.898,284.992,417.209,176.564,22.738,153.556
C00718=1087.891,284.744,417.238,176.561,22.735,153.556
C00719=1087.887,284.496,417.268,176.558,22.732,153.556
C00720=1087.881,284.248,417.298,176.555,22.729,153.555
C00721=1087.875,284.000,417.327,176.552,22.725,153.555
C00722=1087.869,283.752,417.357,176.549,22.722,153.555
C00723=1087.863,283.503,417.386,176.546,22.719,153.555
C00724=1087.858,283.255,417.416,176.543,22.717,153.554
C00725=1087.852,283.007,417.445,176.540,22.713,153.554
C00726=1087.847,282.759,417.474,176.537,22.710,153.554
C00727=1087.841,282.510,417.504,176.534,22.707,153.554
C00728=1087.835,282.262,417.533,176.531,22.704,153.553
C00729=1087.830,282.014,417.563,176.528,22.701,153.553
C00730=1087.825,281.766,417.592,176.525,22.697,153.553
C00731=1087.818,281.518,417.621,176.522,22.694,153.552
C00732=1087.813,281.270,417.650,176.520,22.691,153.552
C00733=1087.807,281.021,417.680,176.517,22.688,153.552
C00734=1087.801,280.773,417.709,176.514,22.685,153.552
C00735=1087.795,280.526,417.738,176.511,22.682,153.551
C00736=1087.790,280.277,417.767,176.508,22.679,153.551
C00737=1087.784,280.029,417.796,176.505,22.676,153.551
C00738=1087.779,279.780,417.825,176.502,22.673,153.551
C00739=1087.772,279.532,417.854,176.499,22.670,153.550
C00740=1087.767,279.284,417.884,176.497,22.667,153.550
C00741=1087.761,279.036,417.913,176.494,22.664,153.550
C00742=1087.756,278.787,417.942,176.491,22.661,153.550
C00743=1087.749,278.539,417.971,176.488,22.658,153.549
C00744=1087.745,278.291,418.000,176.485,22.654,153.549
C00745=1087.738,278.043,418.029,176.482,22.651,153.549
C00746=1087.733,277.794,418.059,176.480,22.648,153.548
C00747=1087.727,277.547,418.087,176.476,22.646,153.548
C00748=1087.722,277.298,418.116,176.474,22.642,153.548
C00749=1087.716,277.050,418.145,176.471,22.639,153.548
C00750=1087.707,276.674,418.189,176.466,22.635,153.547
C00751=1087.699,276.299,418.233,176.461,22.630,153.547
C00752=1087.690,275.923,418.277,176.458,22.626,153.547
C00753=1087.682,275.547,418.320,176.453,22.621,153.546
C00754=1087.676,275.299,418.350,176.450,22.618,153.546
C00755=1087.670,275.050,418.378,176.447,22.615,153.546
C00756=1087.664,274.803,418.407,176.444,22.612,153.545
C00757=1087.659,274.554,418.436,176.441,22.609,153.545
C00758=1087.653,274.306,418.465,176.439,22.606,153.545
C00759=1087.647,274.058,418.493,176.436,22.603,153.545
C00760=1087.642,273.809,418.522,176.433,22.600,153.544
C00761=1087.636,273.561,418.551,176.430,22.597,153.544
C00762=1087.631,273.313,418.579,176.427,22.594,153.544
C00763=1087.624,273.065,418.608,176.424,22.591,153.544
C00764=1087.620,272.816,418.637,176.422,22.588,153.543
C00765=1087.614,272.568,418.665,176.419,22.585,153.543
C00766=1087.607,272.320,418.694,176.415,22.582,153.543
C00767=1087.602,272.072,418.722,176.412,22.579,153.543
C00768=1087.597,271.823,418.752,176.409,22.576,153.542
C00769=1087.591,271.574,418.780,176.407,22.573,153.542
C00770=1087.585,271.327,418.809,176.404,22.570,153.542
C00771=1087.579,271.078,418.837,176.401,22.567,153.542
C00772=1087.574,270.830,418.865,176.398,22.564,153.542
C00773=1087.567,270.582,418.894,176.395,22.561,153.541
C00774=1087.562,270.333,418.923,176.393,22.558,153.541
C00775=1087.557,270.085,418.951,176.390,22.555,153.541
C00776=1087.551,269.837,418.980,176.387,22.552,153.540
C00777=1087.545,269.589,419.008,176.384,22.549,153.540
C00778=1087.539,269.340,419.036,176.381,22.546,153.540
C00779=1087.534,269.092,419.064,176.378,22.544,153.540
C00780=1087.528,268.844,419.093,176.375,22.540,153.540
C00781=1087.522,268.595,419.122,176.373,22.537,153.539
C00782=1087.517,268.347,419.150,176.369,22.534,153.539
C00783=1087.511,268.098,419.178,176.366,22.531,153.539
C00784=1087.506,267.850,419.207,176.364,22.529,153.539
C00785=1087.500,267.602,419.236,176.361,22.526,153.538
C00786=1087.494,267.354,419.264,176.358,22.523,153.538
C00787=1087.488,267.105,419.292,176.355,22.520,153.538
C00788=1087.483,266.857,419.320,176.353,22.517,153.538
C00789=1087.477,266.608,419.348,176.350,22.514,153.538
C00790=1087.472,266.360,419.376,176.347,22.511,153.537
C00791=1087.466,266.112,419.405,176.344,22.508,153.537
C00792=1087.460,265.864,419.433,176.341,22.505,153.537
C00793=1087.454,265.615,419.462,176.338,22.502,153.537
C00794=1087.449,265.367,419.489,176.335,22.499,153.536
C00795=1087.443,265.118,419.518,176.332,22.496,153.536
C00796=1087.438,264.870,419.546,176.329,22.493,153.536
C00797=1087.432,264.622,419.574,176.327,22.490,153.536
C00798=1087.426,264.373,419.602,176.324,22.488,153.535
C00799=1087.420,264.125,419.630,176.321,22.484,153.535
C00800=1087.414,263.877,419.658,176.318,22.482,153.535
C00801=1087.408,263.628,419.686,176.316,22.479,153.535
C00802=1087.400,263.255,419.727,176.311,22.475,153.535
C00803=1087.392,262.882,419.770,176.307,22.470,153.534
C00804=1087.383,262.510,419.812,176.303,22.466,153.534
C00805=1087.374,262.138,419.854,176.298,22.462,153.534
C00806=1087.368,261.888,419.881,176.295,22.459,153.533
C00807=1087.362,261.640,419.909,176.293,22.456,153.533
C00808=1087.356,261.392,419.937,176.290,22.453,153.533
C00809=1087.351,261.144,419.965,176.287,22.450,153.533
C00810=1087.345,260.895,419.993,176.284,22.447,153.533
C00811=1087.339,260.647,420.021,176.281,22.445,153.532
C00812=1087.333,260.398,420.048,176.278,22.442,153.532
C00813=1087.328,260.150,420.076,176.275,22.439,153.532
C00814=1087.322,259.902,420.103,176.273,22.436,153.532
C00815=1087.316,259.653,420.132,176.270,22.434,153.531
C00816=1087.311,259.405,420.159,176.267,22.431,153.531
C00817=1087.304,259.156,420.187,176.264,22.428,153.531
C00818=1087.299,258.908,420.215,176.262,22.425,153.531
C00819=1087.294,258.659,420.242,176.259,22.422,153.531
C00820=1087.287,258.411,420.270,176.256,22.419,153.530
C00821=1087.282,258.163,420.298,176.253,22.416,153.530
C00822=1087.277,257.914,420.325,176.250,22.414,153.530
C00823=1087.270,257.666,420.353,176.247,22.411,153.530
C00824=1087.265,257.418,420.381,176.244,22.408,153.530
C00825=1087.259,257.169,420.408,176.242,22.405,153.529
C00826=1087.253,256.921,420.436,176.239,22.402,153.529
C00827=1087.248,256.672,420.463,176.236,22.399,153.529
C00828=1087.242,256.424,420.490,176.233,22.396,153.529
C00829=1087.236,256.175,420.518,176.231,22.394,153.529
C00830=1087.231,255.927,420.546,176.227,22.391,153.528
C00831=1087.225,255.679,420.573,176.224,22.388,153.528
C00832=1087.219,255.430,420.601,176.222,22.385,153.528
C00833=1087.213,255.182,420.628,176.219,22.382,153.528
C00834=1087.208,254.933,420.655,176.216,22.379,153.528
C00835=1087.202,254.684,420.682,176.214,22.377,153.527
C00836=1087.197,254.436,420.710,176.211,22.374,153.527
C00837=1087.192,254.187,420.738,176.208,22.371,153.527
C00838=1087.185,253.940,420.765,176.206,22.368,153.527
C00839=1087.180,253.690,420.793,176.202,22.365,153.526
C00840=1087.174,253.443,420.820,176.200,22.362,153.526
C00841=1087.169,253.194,420.847,176.196,22.359,153.526
C00842=1087.163,252.946,420.874,176.194,22.357,153.526
C00843=1087.158,252.698,420.902,176.191,22.354,153.526
C00844=1087.151,252.448,420.929,176.188,22.351,153.525
C00845=1087.146,252.200,420.956,176.186,22.348,153.525
C00846=1087.141,251.952,420.984,176.183,22.345,153.525
C00847=1087.135,251.703,421.011,176.180,22.342,153.525
C00848=1087.130,251.455,421.038,176.178,22.340,153.525
C00849=1087.123,251.206,421.066,176.175,22.337,153.524
C00850=1087.118,250.958,421.093,176.171,22.334,153.524
C00851=1087.113,250.709,421.119,176.169,22.331,153.524
C00852=1087.107,250.461,421.147,176.166,22.328,153.524
C00853=1087.101,250.213,421.174,176.163,22.325,153.524
C00854=1087.093,249.837,421.215,176.159,22.321,153.523
C00855=1087.085,249.461,421.256,176.155,22.317,153.523
C00856=1087.076,249.085,421.297,176.151,22.313,153.523
C00857=1087.068,248.710,421.337,176.147,22.308,153.522
C00858=1087.063,248.461,421.365,176.144,22.305,153.522
C00859=1087.057,248.213,421.391,176.141,22.303,153.522
C00860=1087.052,247.964,421.419,176.138,22.299,153.521
C00861=1087.046,247.716,421.446,176.136,22.297,153.521
C00862=1087.040,247.468,421.473,176.133,22.294,153.521
C00863=1087.035,247.219,421.500,176.130,22.291,153.521
C00864=1087.029,246.970,421.527,176.128,22.289,153.521
C00865=1087.023,246.722,421.554,176.125,22.285,153.520
C00866=1087.018,246.473,421.581,176.122,22.283,153.520
C00867=1087.012,246.225,421.607,176.119,22.280,153.520
C00868=1087.006,245.976,421.634,176.116,22.277,153.520
C00869=1087.001,245.728,421.661,176.113,22.274,153.520
C00870=1086.996,245.479,421.688,176.111,22.272,153.520
C00871=1086.990,245.231,421.715,176.108,22.269,153.519
C00872=1086.984,244.983,421.741,176.106,22.266,153.519
C00873=1086.978,244.734,421.768,176.103,22.263,153.519
C00874=1086.973,244.485,421.794,176.100,22.260,153.519
C00875=1086.968,244.237,421.821,176.097,22.258,153.519
C00876=1086.962,243.988,421.848,176.095,22.255,153.518
C00877=1086.956,243.739,421.875,176.091,22.252,153.518
C00878=1086.951,243.490,421.902,176.089,22.250,153.518
C00879=1086.945,243.242,421.929,176.086,22.246,153.518
C00880=1086.939,242.994,421.955,176.084,22.244,153.517
C00881=1086.933,242.745,421.981,176.081,22.241,153.517
C00882=1086.928,242.496,422.008,176.078,22.238,153.517
C00883=1086.922,242.248,422.035,176.076,22.236,153.517
C00884=1086.916,242.000,422.061,176.072,22.233,153.517
C00885=1086.910,241.751,422.088,176.069,22.230,153.517
C00886=1086.905,241.502,422.114,176.067,22.227,153.516
C00887=1086.899,241.254,422.140,176.064,22.224,153.516
C00888=1086.893,241.006,422.167,176.062,22.222,153.516
C00889=1086.888,240.757,422.194,176.059,22.219,153.516
C00890=1086.883,240.508,422.220,176.056,22.216,153.516
C00891=1086.877,240.260,422.247,176.054,22.214,153.515
C00892=1086.871,240.011,422.274,176.050,22.211,153.515
C00893=1086.866,239.762,422.299,176.048,22.208,153.515
C00894=1086.860,239.514,422.326,176.045,22.205,153.515
C00895=1086.854,239.266,422.352,176.042,22.202,153.515
C00896=1086.848,239.017,422.378,176.040,22.200,153.514
C00897=1086.842,238.769,422.405,176.037,22.197,153.514
C00898=1086.837,238.520,422.431,176.035,22.195,153.514
C00899=1086.831,238.271,422.457,176.031,22.192,153.514
C00900=1086.825,238.023,422.484,176.029,22.188,153.514
C00901=1086.820,237.774,422.510,176.026,22.186,153.514
C00902=1086.814,237.525,422.537,176.023,22.183,153.513
C00903=1086.809,237.277,422.562,176.021,22.181,153.513
C00904=1086.803,237.029,422.589,176.018,22.178,153.513
C00905=1086.798,236.780,422.615,176.016,22.175,153.513
C00906=1086.788,236.397,422.655,176.011,22.171,153.512
C00907=1086.781,236.014,422.696,176.007,22.167,153.512
C00908=1086.772,235.632,422.736,176.003,22.162,153.512
C00909=1086.763,235.250,422.776,175.999,22.159,153.512
C00910=1086.757,235.001,422.802,175.996,22.155,153.511
C00911=1086.752,234.753,422.828,175.993,22.153,153.511
C00912=1086.746,234.504,422.854,175.991,22.150,153.511
C00913=1086.741,234.255,422.880,175.988,22.147,153.511
C00914=1086.736,234.007,422.907,175.985,22.145,153.511
C00915=1086.730,233.758,422.932,175.982,22.142,153.510
C00916=1086.724,233.510,422.958,175.980,22.139,153.510
C00917=1086.718,233.261,422.984,175.977,22.136,153.510
C00918=1086.713,233.012,423.010,175.975,22.134,153.510
C00919=1086.707,232.763,423.036,175.972,22.131,153.510
C00920=1086.701,232.515,423.062,175.969,22.128,153.510
C00921=1086.696,232.267,423.088,175.967,22.125,153.509
C00922=1086.690,232.018,423.114,175.963,22.123,153.509
C00923=1086.685,231.769,423.140,175.961,22.120,153.509
C00924=1086.678,231.521,423.166,175.958,22.117,153.509
C00925=1086.673,231.272,423.192,175.956,22.115,153.509
C00926=1086.668,231.023,423.217,175.953,22.112,153.508
C00927=1086.663,230.774,423.243,175.951,22.110,153.508
C00928=1086.656,230.526,423.269,175.948,22.106,153.508
C00929=1086.651,230.277,423.295,175.945,22.104,153.508
C00930=1086.645,230.028,423.321,175.942,22.101,153.508
C00931=1086.640,229.780,423.346,175.939,22.098,153.508
C00932=1086.634,229.531,423.372,175.937,22.096,153.507
C00933=1086.628,229.283,423.397,175.934,22.093,153.507
C00934=1086.622,229.034,423.423,175.932,22.090,153.507
C00935=1086.617,228.785,423.449,175.929,22.088,153.507
C00936=1086.611,228.537,423.475,175.926,22.085,153.507
C00937=1086.606,228.288,423.501,175.923,22.082,153.507
C00938=1086.599,228.040,423.526,175.921,22.080,153.506
C00939=1086.594,227.791,423.552,175.918,22.077,153.506
C00940=1086.588,227.543,423.577,175.916,22.074,153.506
C00941=1086.583,227.294,423.603,175.913,22.072,153.506
C00942=1086.577,227.045,423.628,175.911,22.069,153.505
C00943=1086.571,226.796,423.654,175.908,22.066,153.505
C00944=1086.566,226.548,423.679,175.905,22.064,153.505
C00945=1086.560,226.299,423.705,175.902,22.061,153.505
C00946=1086.554,226.051,423.731,175.900,22.059,153.505
C00947=1086.549,225.802,423.756,175.897,22.055,153.505
C00948=1086.543,225.554,423.781,175.895,22.053,153.504
C00949=1086.538,225.304,423.807,175.892,22.050,153.504
C00950=1086.531,225.055,423.832,175.889,22.048,153.504
C00951=1086.527,224.807,423.858,175.886,22.044,153.504
C00952=1086.520,224.558,423.883,175.884,22.042,153.504
C00953=1086.515,224.309,423.909,175.881,22.039,153.504
C00954=1086.509,224.062,423.934,175.879,22.037,153.503
C00955=1086.504,223.813,423.960,175.876,22.034,153.503
C00956=1086.498,223.565,423.985,175.874,22.031,153.503
C00957=1086.493,223.315,424.010,175.871,22.029,153.503
C00958=1086.484,222.924,424.049,175.867,22.024,153.502
C00959=1086.475,222.533,424.090,175.862,22.020,153.502
C00960=1086.466,222.142,424.130,175.859,22.016,153.502
C00961=1086.457,221.751,424.169,175.854,22.012,153.502
C00962=1086.452,221.502,424.195,175.852,22.009,153.501
C00963=1086.446,221.254,424.220,175.849,22.006,153.501
C00964=1086.440,221.004,424.244,175.847,22.004,153.501
C00965=1086.435,220.755,424.270,175.843,22.001,153.501
C00966=1086.429,220.507,424.295,175.841,21.999,153.501
C00967=1086.423,220.258,424.320,175.838,21.996,153.501
C00968=1086.418,220.010,424.345,175.836,21.993,153.500
C00969=1086.412,219.761,424.371,175.833,21.990,153.500
C00970=1086.406,219.512,424.395,175.831,21.988,153.500
C00971=1086.401,219.264,424.420,175.828,21.985,153.500
C00972=1086.395,219.015,424.446,175.825,21.983,153.500
C00973=1086.390,218.766,424.471,175.823,21.980,153.499
C00974=1086.384,218.518,424.496,175.820,21.977,153.499
C00975=1086.378,218.268,424.520,175.818,21.975,153.499
C00976=1086.372,218.020,424.545,175.815,21.972,153.499
C00977=1086.366,217.771,424.570,175.812,21.969,153.499
C00978=1086.362,217.523,424.596,175.810,21.966,153.499
C00979=1086.355,217.274,424.621,175.807,21.964,153.498
C00980=1086.350,217.026,424.645,175.804,21.961,153.498
C00981=1086.344,216.776,424.670,175.802,21.959,153.498
C00982=1086.339,216.528,424.695,175.800,21.956,153.498
C00983=1086.333,216.279,424.720,175.797,21.953,153.498
C00984=1086.328,216.031,424.745,175.795,21.951,153.498
C00985=1086.322,215.782,424.770,175.791,21.948,153.497
C00986=1086.316,215.534,424.795,175.789,21.945,153.497
C00987=1086.310,215.284,424.819,175.786,21.942,153.497
C00988=1086.305,215.036,424.844,175.784,21.940,153.497
C00989=1086.300,214.787,424.869,175.781,21.937,153.497
C00990=1086.294,214.538,424.894,175.779,21.935,153.497
C00991=1086.288,214.289,424.919,175.776,21.932,153.496
C00992=1086.283,214.041,424.943,175.774,21.929,153.496
C00993=1086.278,213.792,424.968,175.771,21.927,153.496
C00994=1086.271,213.544,424.993,175.768,21.924,153.496
C00995=1086.266,213.295,425.017,175.766,21.922,153.496
C00996=1086.260,213.046,425.042,175.763,21.918,153.495
C00997=1086.255,212.798,425.067,175.761,21.916,153.495
C00998=1086.249,212.548,425.091,175.759,21.913,153.495
C00999=1086.243,212.300,425.116,175.755,21.911,153.495
C01000=1086.237,212.051,425.140,175.753,21.908,153.495
C01001=1086.232,211.803,425.165,175.750,21.905,153.495
C01002=1086.227,211.554,425.189,175.748,21.903,153.494
C01003=1086.221,211.305,425.214,175.745,21.900,153.494
C01004=1086.215,211.056,425.238,175.743,21.898,153.494
C01005=1086.209,210.807,425.264,175.740,21.895,153.494
C01006=1086.204,210.559,425.288,175.738,21.892,153.494
C01007=1086.199,210.310,425.312,175.735,21.889,153.493
C01008=1086.193,210.061,425.337,175.732,21.887,153.493
C01009=1086.187,209.812,425.361,175.730,21.884,153.493
C01010=1086.179,209.425,425.400,175.726,21.880,153.493
C01011=1086.170,209.038,425.437,175.722,21.876,153.493
C01012=1086.160,208.651,425.475,175.718,21.872,153.492
C01013=1086.153,208.264,425.514,175.714,21.868,153.492
C01014=1086.130,207.237,425.612,175.634,21.826,153.495
C01015=1086.123,206.988,425.636,175.631,21.824,153.495
C01016=1086.118,206.739,425.660,175.629,21.823,153.496
C01017=1086.112,206.490,425.685,175.626,21.821,153.496
C01018=1086.107,206.241,425.708,175.624,21.819,153.495
C01019=1086.101,205.993,425.732,175.620,21.817,153.496
C01020=1086.095,205.744,425.756,175.618,21.816,153.496
C01021=1086.090,205.495,425.779,175.615,21.814,153.496
C01022=1086.084,205.246,425.804,175.613,21.812,153.496
C01023=1086.078,204.998,425.827,175.610,21.811,153.496
C01024=1086.073,204.749,425.851,175.608,21.809,153.496
C01025=1086.068,204.500,425.875,175.604,21.807,153.496
C01026=1086.062,204.250,425.898,175.602,21.805,153.496
C01027=1086.056,204.002,425.923,175.599,21.804,153.496
C01028=1086.050,203.754,425.946,175.597,21.802,153.496
C01029=1086.045,203.504,425.970,175.594,21.800,153.496
C01030=1086.040,203.256,425.994,175.592,21.798,153.496
C01031=1086.034,203.007,426.017,175.589,21.797,153.496
C01032=1086.029,202.758,426.041,175.586,21.795,153.496
C01033=1086.023,202.509,426.064,175.583,21.793,153.496
C01034=1086.017,202.260,426.089,175.581,21.792,153.496
C01035=1086.012,202.011,426.112,175.578,21.790,153.496
C01036=1086.006,201.763,426.136,175.576,21.788,153.496
C01037=1086.001,201.514,426.159,175.573,21.787,153.496
C01038=1085.995,201.265,426.183,175.571,21.785,153.496
C01039=1085.990,201.016,426.206,175.568,21.784,153.496
C01040=1085.984,200.768,426.230,175.565,21.781,153.496
C01041=1085.977,200.518,426.253,175.562,21.780,153.497
C01042=1085.972,200.270,426.277,175.560,21.778,153.497
C01043=1085.966,200.021,426.300,175.557,21.777,153.497
C01044=1085.960,199.773,426.324,175.555,21.775,153.497
C01045=1085.955,199.523,426.348,175.552,21.773,153.497
C01046=1085.950,199.275,426.371,175.550,21.772,153.497
C01047=1085.944,199.026,426.394,175.547,21.770,153.497
C01048=1085.939,198.777,426.418,175.544,21.768,153.497
C01049=1085.933,198.528,426.441,175.541,21.766,153.497
C01050=1085.927,198.280,426.464,175.539,21.765,153.497
C01051=1085.922,198.031,426.488,175.536,21.763,153.497
C01052=1085.915,197.781,426.511,175.533,21.762,153.497
C01053=1085.909,197.533,426.535,175.531,21.760,153.497
C01054=1085.904,197.284,426.558,175.528,21.758,153.497
C01055=1085.899,197.035,426.581,175.526,21.757,153.497
C01056=1085.893,196.786,426.605,175.524,21.755,153.497
C01057=1085.887,196.538,426.628,175.521,21.753,153.497
C01058=1085.882,196.288,426.652,175.518,21.751,153.497
C01059=1085.876,196.039,426.674,175.515,21.750,153.497
C01060=1085.870,195.791,426.697,175.513,21.748,153.497
C01061=1085.865,195.542,426.722,175.510,21.746,153.497
C01062=1085.859,195.293,426.745,175.507,21.745,153.497
C01063=1085.854,195.044,426.768,175.505,21.743,153.497
C01064=1085.848,194.795,426.791,175.502,21.741,153.498
C01065=1085.843,194.546,426.814,175.500,21.740,153.497
C01066=1085.837,194.298,426.838,175.497,21.738,153.498
C01067=1085.831,194.049,426.861,175.495,21.736,153.498
C01068=1085.825,193.800,426.884,175.493,21.734,153.498
C01069=1085.820,193.551,426.907,175.490,21.733,153.498
C01070=1085.815,193.302,426.930,175.487,21.731,153.498
C01071=1085.809,193.053,426.953,175.484,21.729,153.498
C01072=1085.804,192.805,426.976,175.482,21.728,153.498
C01073=1085.799,192.556,426.999,175.479,21.726,153.498
C01074=1085.793,192.307,427.023,175.476,21.724,153.498
C01075=1085.787,192.029,427.048,175.474,21.722,153.498
C01076=1085.780,191.750,427.074,175.471,21.720,153.498
C01077=1085.774,191.472,427.100,175.468,21.718,153.498
C01078=1085.768,191.194,427.126,175.466,21.717,153.498
C01079=1085.762,190.945,427.149,175.463,21.715,153.498
C01080=1085.757,190.697,427.171,175.461,21.713,153.498
C01081=1085.752,190.448,427.195,175.457,21.711,153.498
C01082=1085.746,190.199,427.218,175.455,21.710,153.498
C01083=1085.740,189.950,427.241,175.452,21.708,153.498
C01084=1085.735,189.701,427.264,175.450,21.706,153.498
C01085=1085.729,189.452,427.287,175.447,21.704,153.498
C01086=1085.724,189.203,427.310,175.445,21.703,153.498
C01087=1085.718,188.954,427.333,175.443,21.701,153.498
C01088=1085.713,188.706,427.355,175.440,21.699,153.498
C01089=1085.708,188.457,427.378,175.437,21.697,153.498
C01090=1085.702,188.208,427.401,175.435,21.696,153.498
C01091=1085.696,187.959,427.424,175.432,21.694,153.498
C01092=1085.690,187.710,427.447,175.430,21.692,153.498
C01093=1085.686,187.461,427.470,175.428,21.691,153.498
C01094=1085.680,187.213,427.493,175.425,21.689,153.498
C01095=1085.675,186.964,427.516,175.423,21.687,153.498
C01096=1085.669,186.714,427.538,175.420,21.685,153.498
C01097=1085.663,186.465,427.561,175.418,21.684,153.498
C01098=1085.658,186.217,427.584,175.415,21.682,153.498
C01099=1085.653,185.968,427.606,175.413,21.680,153.498
C01100=1085.647,185.719,427.629,175.410,21.678,153.498
C01101=1085.642,185.469,427.652,175.408,21.677,153.498
C01102=1085.637,185.221,427.675,175.405,21.675,153.498
C01103=1085.631,184.972,427.698,175.403,21.673,153.498
C01104=1085.625,184.724,427.720,175.400,21.671,153.498
C01105=1085.619,184.474,427.742,175.398,21.670,153.499
C01106=1085.614,184.225,427.765,175.395,21.668,153.499
C01107=1085.608,183.976,427.788,175.393,21.667,153.499
C01108=1085.602,183.727,427.810,175.390,21.665,153.499
C01109=1085.597,183.479,427.832,175.388,21.664,153.499
C01110=1085.591,183.230,427.855,175.385,21.662,153.499
C01111=1085.585,182.981,427.878,175.383,21.660,153.499
C01112=1085.580,182.732,427.901,175.380,21.659,153.499
C01113=1085.573,182.483,427.923,175.378,21.657,153.499
C01114=1085.568,182.234,427.945,175.375,21.655,153.499
C01115=1085.562,181.985,427.968,175.373,21.653,153.499
C01116=1085.556,181.737,427.990,175.370,21.652,153.499
C01117=1085.551,181.487,428.012,175.368,21.650,153.499
C01118=1085.545,181.238,428.035,175.365,21.648,153.499
C01119=1085.540,180.989,428.058,175.362,21.647,153.499
C01120=1085.533,180.740,428.080,175.360,21.645,153.499
C01121=1085.528,180.492,428.102,175.357,21.644,153.499
C01122=1085.523,180.243,428.125,175.355,21.642,153.499
C01123=1085.516,179.994,428.147,175.353,21.640,153.499
C01124=1085.511,179.744,428.169,175.350,21.639,153.499
C01125=1085.506,179.496,428.192,175.348,21.637,153.499
C01126=1085.499,179.247,428.213,175.345,21.635,153.499
C01127=1085.494,178.998,428.236,175.342,21.634,153.499
C01128=1085.488,178.749,428.259,175.340,21.632,153.499
C01129=1085.483,178.500,428.281,175.337,21.630,153.500
C01130=1085.477,178.251,428.303,175.335,21.629,153.500
C01131=1085.471,178.002,428.326,175.333,21.627,153.499
C01132=1085.466,177.753,428.348,175.331,21.626,153.500
C01133=1085.460,177.504,428.369,175.328,21.624,153.500
C01134=1085.455,177.255,428.392,175.326,21.622,153.500
C01135=1085.448,177.006,428.414,175.323,21.621,153.500
C01136=1085.443,176.757,428.437,175.321,21.619,153.500
C01137=1085.438,176.509,428.459,175.319,21.617,153.500
C01138=1085.432,176.259,428.480,175.316,21.616,153.500
C01139=1085.425,175.981,428.505,175.313,21.614,153.500
C01140=1085.419,175.703,428.530,175.310,21.611,153.500
C01141=1085.413,175.424,428.555,175.308,21.609,153.500
C01142=1085.406,175.146,428.580,175.305,21.608,153.500
C01143=1085.401,174.896,428.602,175.303,21.606,153.500
C01144=1085.396,174.648,428.624,175.300,21.604,153.500
C01145=1085.390,174.399,428.646,175.298,21.603,153.500
C01146=1085.384,174.149,428.668,175.295,21.601,153.500
C01147=1085.378,173.901,428.690,175.293,21.599,153.500
C01148=1085.373,173.652,428.712,175.290,21.597,153.500
C01149=1085.368,173.403,428.734,175.288,21.596,153.500
C01150=1085.362,173.154,428.756,175.285,21.594,153.500
C01151=1085.356,172.905,428.779,175.283,21.592,153.500
C01152=1085.351,172.657,428.800,175.280,21.590,153.500
C01153=1085.345,172.407,428.822,175.279,21.589,153.500
C01154=1085.341,172.158,428.844,175.277,21.587,153.500
C01155=1085.334,171.910,428.867,175.274,21.586,153.500
C01156=1085.329,171.660,428.889,175.271,21.584,153.500
C01157=1085.323,171.412,428.910,175.269,21.582,153.500
C01158=1085.318,171.162,428.932,175.267,21.580,153.500
C01159=1085.312,170.914,428.954,175.264,21.578,153.500
C01160=1085.307,170.664,428.976,175.262,21.577,153.500
C01161=1085.301,170.416,428.997,175.259,21.575,153.500
C01162=1085.295,170.167,429.020,175.257,21.573,153.500
C01163=1085.289,169.917,429.042,175.254,21.571,153.500
C01164=1085.284,169.669,429.064,175.253,21.570,153.500
C01165=1085.279,169.419,429.086,175.250,21.569,153.500
C01166=1085.273,169.171,429.107,175.248,21.567,153.500
C01167=1085.268,168.921,429.129,175.245,21.565,153.500
C01168=1085.262,168.673,429.151,175.243,21.563,153.500
C01169=1085.257,168.423,429.173,175.240,21.561,153.500
C01170=1085.251,168.175,429.194,175.238,21.559,153.500
C01171=1085.246,167.925,429.216,175.236,21.557,153.500
C01172=1085.240,167.677,429.238,175.233,21.556,153.500
C01173=1085.235,167.427,429.260,175.231,21.555,153.500
C01174=1085.229,167.179,429.281,175.229,21.553,153.500
C01175=1085.224,166.929,429.303,175.227,21.551,153.500
C01176=1085.218,166.681,429.325,175.224,21.549,153.500
C01177=1085.212,166.431,429.346,175.222,21.547,153.500
C01178=1085.207,166.183,429.368,175.219,21.545,153.500
C01179=1085.202,165.934,429.389,175.217,21.543,153.500
C01180=1085.196,165.684,429.412,175.214,21.541,153.500
C01181=1085.191,165.436,429.433,175.213,21.541,153.500
C01182=1085.186,165.186,429.455,175.210,21.539,153.500
C01183=1085.180,164.938,429.476,175.208,21.537,153.500
C01184=1085.175,164.688,429.499,175.205,21.535,153.500
C01185=1085.169,164.440,429.520,175.203,21.533,153.500
C01186=1085.164,164.191,429.541,175.201,21.531,153.500
C01187=1085.158,163.941,429.563,175.198,21.529,153.500
C01188=1085.153,163.693,429.584,175.196,21.527,153.500
C01189=1085.147,163.443,429.606,175.194,21.526,153.500
C01190=1085.142,163.195,429.627,175.192,21.524,153.500
C01191=1085.137,162.946,429.649,175.189,21.522,153.500
C01192=1085.131,162.696,429.670,175.187,21.520,153.500
C01193=1085.126,162.447,429.692,175.185,21.519,153.500
C01194=1085.121,162.199,429.713,175.182,21.517,153.500
C01195=1085.114,161.950,429.735,175.180,21.515,153.500
C01196=1085.110,161.701,429.757,175.178,21.513,153.500
C01197=1085.104,161.451,429.778,175.176,21.512,153.500
C01198=1085.098,161.202,429.799,175.173,21.510,153.500
C01199=1085.093,160.954,429.820,175.171,21.508,153.500
C01200=1085.087,160.704,429.842,175.168,21.506,153.500
C01201=1085.082,160.455,429.863,175.166,21.505,153.500
C01202=1085.076,160.206,429.885,175.164,21.503,153.500
C01203=1085.069,159.927,429.908,175.161,21.501,153.500
C01204=1085.063,159.648,429.932,175.159,21.499,153.500
C01205=1085.057,159.369,429.956,175.156,21.497,153.500
C01206=1085.051,159.091,429.979,175.154,21.495,153.500
C01207=1085.045,158.842,430.001,175.151,21.493,153.500
C01208=1085.040,158.593,430.022,175.149,21.491,153.500
C01209=1085.034,158.344,430.044,175.147,21.490,153.500
C01210=1085.029,158.095,430.065,175.145,21.489,153.500
C01211=1085.023,157.846,430.086,175.142,21.487,153.500
C01212=1085.017,157.597,430.107,175.140,21.485,153.500
C01213=1085.012,157.348,430.128,175.137,21.483,153.500
C01214=1085.006,157.099,430.149,175.135,21.481,153.500
C01215=1085.000,156.850,430.171,175.133,21.479,153.500
C01216=1084.995,156.601,430.191,175.131,21.478,153.500
C01217=1084.989,156.352,430.213,175.129,21.476,153.500
C01218=1084.984,156.102,430.234,175.126,21.474,153.500
C01219=1084.978,155.854,430.255,175.124,21.472,153.500
C01220=1084.973,155.605,430.276,175.121,21.470,153.500
C01221=1084.967,155.355,430.298,175.120,21.469,153.500
C01222=1084.962,155.106,430.318,175.117,21.467,153.500
C01223=1084.957,154.858,430.339,175.115,21.465,153.500
C01224=1084.951,154.608,430.360,175.112,21.464,153.500
C01225=1084.944,154.360,430.381,175.110,21.462,153.500
C01226=1084.939,154.111,430.402,175.108,21.461,153.500
C01227=1084.933,153.861,430.423,175.106,21.459,153.500
C01228=1084.928,153.612,430.444,175.104,21.457,153.500
C01229=1084.922,153.364,430.465,175.101,21.455,153.500
C01230=1084.916,153.114,430.486,175.099,21.453,153.500
C01231=1084.911,152.865,430.506,175.097,21.452,153.500
C01232=1084.905,152.616,430.528,175.095,21.450,153.500
C01233=1084.900,152.366,430.549,175.092,21.448,153.500
C01234=1084.894,152.118,430.570,175.090,21.446,153.500
C01235=1084.889,151.869,430.590,175.088,21.444,153.500
C01236=1084.884,151.620,430.611,175.086,21.443,153.499
C01237=1084.877,151.370,430.633,175.084,21.441,153.499
C01238=1084.872,151.121,430.653,175.081,21.439,153.499
C01239=1084.867,150.872,430.674,175.079,21.437,153.499
C01240=1084.861,150.624,430.695,175.077,21.436,153.499
C01241=1084.855,150.374,430.716,175.075,21.434,153.499
C01242=1084.849,150.125,430.736,175.072,21.432,153.499
C01243=1084.844,149.877,430.757,175.070,21.430,153.499
C01244=1084.839,149.627,430.778,175.068,21.428,153.499
C01245=1084.833,149.378,430.799,175.066,21.427,153.499
C01246=1084.827,149.129,430.820,175.064,21.425,153.499
C01247=1084.822,148.880,430.840,175.061,21.423,153.499
C01248=1084.817,148.631,430.861,175.059,21.421,153.499
C01249=1084.811,148.382,430.881,175.057,21.420,153.499
C01250=1084.805,148.132,430.902,175.055,21.418,153.499
C01251=1084.799,147.884,430.923,175.052,21.416,153.499
C01252=1084.794,147.635,430.944,175.050,21.414,153.499
C01253=1084.789,147.385,430.964,175.048,21.413,153.499
C01254=1084.782,147.136,430.985,175.046,21.411,153.499
C01255=1084.777,146.887,431.005,175.044,21.409,153.499
C01256=1084.771,146.638,431.026,175.041,21.407,153.499
C01257=1084.765,146.390,431.046,175.040,21.406,153.499
C01258=1084.759,146.140,431.067,175.037,21.404,153.499
C01259=1084.754,145.891,431.088,175.035,21.402,153.499
C01260=1084.749,145.641,431.108,175.032,21.400,153.499
C01261=1084.743,145.393,431.128,175.031,21.399,153.499
C01262=1084.738,145.144,431.149,175.028,21.397,153.499
C01263=1084.732,144.895,431.170,175.026,21.395,153.499
C01264=1084.726,144.645,431.191,175.024,21.393,153.499
C01265=1084.720,144.396,431.211,175.022,21.391,153.499
C01266=1084.715,144.147,431.232,175.020,21.390,153.499
C01267=1084.709,143.868,431.254,175.017,21.387,153.499
C01268=1084.703,143.589,431.277,175.015,21.385,153.499
C01269=1084.696,143.311,431.300,175.013,21.383,153.499
C01270=1084.690,143.031,431.323,175.010,21.382,153.499
C01271=1084.684,142.782,431.344,175.008,21.380,153.499
C01272=1084.679,142.533,431.364,175.005,21.378,153.499
C01273=1084.673,142.284,431.384,175.003,21.375,153.499
C01274=1084.668,142.035,431.405,175.002,21.374,153.498
C01275=1084.662,141.785,431.426,174.999,21.372,153.498
C01276=1084.656,141.536,431.446,174.997,21.370,153.498
C01277=1084.651,141.287,431.466,174.994,21.368,153.498
C01278=1084.645,141.039,431.486,174.993,21.367,153.498
C01279=1084.640,140.789,431.507,174.990,21.365,153.498
C01280=1084.635,140.540,431.527,174.988,21.363,153.498
C01281=1084.629,140.291,431.546,174.986,21.361,153.498
C01282=1084.623,140.042,431.567,174.984,21.359,153.498
C01283=1084.617,139.793,431.587,174.982,21.357,153.498
C01284=1084.612,139.543,431.608,174.979,21.356,153.498
C01285=1084.606,139.294,431.628,174.978,21.354,153.498
C01286=1084.600,139.045,431.648,174.976,21.352,153.498
C01287=1084.594,138.796,431.668,174.973,21.350,153.498
C01288=1084.589,138.547,431.689,174.971,21.349,153.498
C01289=1084.583,138.298,431.708,174.969,21.347,153.498
C01290=1084.578,138.049,431.729,174.967,21.345,153.498
C01291=1084.572,137.800,431.749,174.965,21.343,153.498
C01292=1084.567,137.551,431.769,174.963,21.341,153.498
C01293=1084.561,137.302,431.789,174.961,21.340,153.498
C01294=1084.556,137.053,431.810,174.958,21.338,153.498
C01295=1084.550,136.803,431.829,174.957,21.336,153.498
C01296=1084.545,136.554,431.850,174.954,21.334,153.498
C01297=1084.539,136.305,431.869,174.952,21.332,153.498
C01298=1084.533,136.056,431.890,174.950,21.330,153.498
C01299=1084.527,135.806,431.910,174.948,21.329,153.498
C01300=1084.521,135.557,431.930,174.946,21.327,153.498
C01301=1084.516,135.308,431.950,174.943,21.325,153.498
C01302=1084.510,135.059,431.970,174.942,21.323,153.497
C01303=1084.505,134.810,431.990,174.939,21.321,153.497
C01304=1084.499,134.561,432.010,174.937,21.319,153.497
C01305=1084.494,134.312,432.030,174.936,21.318,153.497
C01306=1084.488,134.062,432.050,174.933,21.316,153.497
C01307=1084.482,133.813,432.070,174.931,21.313,153.497
C01308=1084.477,133.564,432.090,174.929,21.312,153.497
C01309=1084.471,133.315,432.109,174.927,21.310,153.497
C01310=1084.466,133.066,432.130,174.925,21.308,153.497
C01311=1084.460,132.817,432.150,174.922,21.306,153.497
C01312=1084.454,132.568,432.169,174.921,21.304,153.497
C01313=1084.449,132.318,432.190,174.918,21.303,153.497
C01314=1084.443,132.069,432.209,174.916,21.301,153.497
C01315=1084.437,131.820,432.229,174.914,21.299,153.497
C01316=1084.431,131.571,432.249,174.912,21.297,153.497
C01317=1084.426,131.322,432.269,174.910,21.295,153.497
C01318=1084.420,131.073,432.289,174.908,21.294,153.497
C01319=1084.415,130.823,432.308,174.906,21.292,153.497
C01320=1084.409,130.575,432.328,174.903,21.290,153.497
C01321=1084.403,130.325,432.347,174.902,21.288,153.497
C01322=1084.398,130.076,432.368,174.900,21.286,153.497
C01323=1084.392,129.827,432.387,174.897,21.284,153.496
C01324=1084.386,129.578,432.407,174.896,21.283,153.496
C01325=1084.380,129.329,432.427,174.893,21.281,153.496
C01326=1084.374,129.080,432.446,174.891,21.279,153.496
C01327=1084.369,128.830,432.465,174.889,21.277,153.496
C01328=1084.363,128.581,432.486,174.887,21.276,153.496
C01329=1084.358,128.332,432.505,174.885,21.273,153.496
C01330=1084.352,128.083,432.525,174.883,21.272,153.496
C01331=1084.345,127.804,432.546,174.881,21.270,153.496
C01332=1084.339,127.524,432.569,174.879,21.267,153.496
C01333=1084.333,127.246,432.590,174.876,21.266,153.496
C01334=1084.326,126.966,432.613,174.874,21.264,153.496
C01335=1084.321,126.717,432.632,174.872,21.261,153.496
C01336=1084.315,126.468,432.652,174.870,21.260,153.496
C01337=1084.310,126.219,432.671,174.868,21.258,153.496
C01338=1084.304,125.970,432.691,174.865,21.256,153.496
C01339=1084.298,125.721,432.710,174.864,21.254,153.496
C01340=1084.293,125.471,432.730,174.862,21.252,153.496
C01341=1084.287,125.222,432.750,174.859,21.250,153.496
C01342=1084.281,124.973,432.769,174.858,21.248,153.495
C01343=1084.276,124.724,432.788,174.855,21.247,153.495
C01344=1084.270,124.475,432.808,174.853,21.245,153.495
C01345=1084.264,124.225,432.828,174.852,21.243,153.495
C01346=1084.259,123.977,432.847,174.849,21.241,153.495
C01347=1084.253,123.728,432.867,174.848,21.239,153.495
C01348=1084.247,123.478,432.886,174.846,21.237,153.495
C01349=1084.241,123.229,432.905,174.843,21.235,153.495
C01350=1084.236,122.980,432.924,174.842,21.234,153.495
C01351=1084.230,122.731,432.944,174.839,21.231,153.495
C01352=1084.225,122.482,432.964,174.837,21.229,153.495
C01353=1084.220,122.232,432.983,174.835,21.228,153.495
C01354=1084.214,121.983,433.002,174.833,21.226,153.495
C01355=1084.208,121.734,433.022,174.831,21.224,153.495
C01356=1084.202,121.485,433.041,174.829,21.222,153.495
C01357=1084.197,121.235,433.061,174.827,21.220,153.494
C01358=1084.192,120.986,433.079,174.826,21.218,153.494
C01359=1084.186,120.737,433.099,174.823,21.217,153.494
C01360=1084.180,120.488,433.118,174.821,21.214,153.494
C01361=1084.174,120.239,433.138,174.819,21.213,153.494
C01362=1084.168,119.989,433.157,174.817,21.210,153.494
C01363=1084.163,119.741,433.176,174.815,21.208,153.494
C01364=1084.158,119.491,433.195,174.813,21.207,153.494
C01365=1084.152,119.242,433.215,174.811,21.205,153.494
C01366=1084.146,118.992,433.234,174.810,21.203,153.494
C01367=1084.141,118.744,433.253,174.807,21.201,153.494
C01368=1084.135,118.495,433.273,174.805,21.199,153.494
C01369=1084.130,118.245,433.292,174.804,21.197,153.493
C01370=1084.124,117.996,433.311,174.801,21.195,153.493
C01371=1084.119,117.747,433.330,174.800,21.193,153.493
C01372=1084.113,117.498,433.349,174.797,21.191,153.493
C01373=1084.107,117.248,433.368,174.795,21.189,153.493
C01374=1084.102,117.000,433.387,174.794,21.187,153.493
C01375=1084.097,116.750,433.407,174.792,21.185,153.493
C01376=1084.091,116.501,433.426,174.790,21.184,153.493
C01377=1084.085,116.251,433.445,174.788,21.181,153.493
C01378=1084.080,116.002,433.464,174.785,21.179,153.493
C01379=1084.074,115.753,433.483,174.784,21.177,153.493
C01380=1084.069,115.504,433.502,174.782,21.175,153.493
C01381=1084.064,115.255,433.521,174.780,21.174,153.492
C01382=1084.058,115.005,433.541,174.778,21.172,153.492
C01383=1084.052,114.756,433.560,174.776,21.169,153.492
C01384=1084.047,114.507,433.579,174.774,21.168,153.492
C01385=1084.041,114.258,433.597,174.772,21.165,153.492
C01386=1084.035,114.009,433.617,174.770,21.164,153.492
C01387=1084.029,113.759,433.636,174.768,21.162,153.492
C01388=1084.024,113.511,433.655,174.766,21.160,153.492
C01389=1084.019,113.261,433.673,174.764,21.158,153.492
C01390=1084.013,113.011,433.692,174.762,21.156,153.492
C01391=1084.007,112.763,433.711,174.761,21.154,153.492
C01392=1084.002,112.513,433.730,174.758,21.152,153.491
C01393=1083.996,112.264,433.749,174.756,21.150,153.491
C01394=1083.990,112.015,433.768,174.755,21.148,153.491
C01395=1083.983,111.736,433.789,174.752,21.146,153.491
C01396=1083.978,111.457,433.811,174.750,21.144,153.491
C01397=1083.971,111.177,433.830,174.748,21.141,153.491
C01398=1083.965,110.898,433.852,174.746,21.140,153.491
C01399=1083.959,110.649,433.871,174.744,21.138,153.491
C01400=1083.954,110.400,433.890,174.742,21.136,153.491
C01401=1083.948,110.151,433.908,174.740,21.134,153.491
C01402=1083.942,109.902,433.928,174.738,21.132,153.491
C01403=1083.937,109.652,433.946,174.736,21.129,153.490
C01404=1083.930,109.402,433.965,174.734,21.128,153.490
C01405=1083.925,109.154,433.984,174.732,21.126,153.490
C01406=1083.920,108.904,434.003,174.731,21.124,153.490
C01407=1083.913,108.655,434.021,174.728,21.122,153.490
C01408=1083.908,108.406,434.040,174.727,21.120,153.490
C01409=1083.902,108.157,434.058,174.725,21.118,153.490
C01410=1083.897,107.907,434.076,174.722,21.116,153.490
C01411=1083.891,107.658,434.096,174.721,21.114,153.490
C01412=1083.885,107.409,434.114,174.719,21.112,153.490
C01413=1083.880,107.160,434.133,174.717,21.110,153.490
C01414=1083.874,106.910,434.151,174.715,21.108,153.490
C01415=1083.868,106.661,434.170,174.714,21.106,153.489
C01416=1083.863,106.412,434.189,174.711,21.105,153.489
C01417=1083.857,106.162,434.207,174.710,21.103,153.489
C01418=1083.852,105.914,434.226,174.707,21.101,153.489
C01419=1083.846,105.664,434.244,174.705,21.098,153.489
C01420=1083.840,105.415,434.263,174.704,21.096,153.489
C01421=1083.835,105.166,434.282,174.701,21.094,153.489
C01422=1083.829,104.916,434.300,174.700,21.093,153.489
C01423=1083.824,104.667,434.319,174.698,21.091,153.489
C01424=1083.817,104.418,434.338,174.696,21.089,153.488
C01425=1083.812,104.169,434.356,174.694,21.086,153.488
C01426=1083.806,103.920,434.374,174.693,21.085,153.488
C01427=1083.801,103.670,434.393,174.691,21.082,153.488
C01428=1083.795,103.421,434.411,174.688,21.081,153.488
C01429=1083.789,103.171,434.430,174.687,21.079,153.488
C01430=1083.784,102.922,434.449,174.685,21.076,153.488
C01431=1083.778,102.673,434.467,174.683,21.075,153.488
C01432=1083.773,102.424,434.485,174.681,21.072,153.488
C01433=1083.767,102.174,434.503,174.679,21.071,153.488
C01434=1083.762,101.926,434.522,174.677,21.068,153.487
C01435=1083.756,101.676,434.540,174.676,21.067,153.487
C01436=1083.751,101.427,434.559,174.673,21.065,153.487
C01437=1083.745,101.177,434.577,174.672,21.063,153.487
C01438=1083.740,100.929,434.596,174.670,21.060,153.487
C01439=1083.733,100.679,434.614,174.668,21.059,153.487
C01440=1083.728,100.430,434.632,174.666,21.056,153.487
C01441=1083.722,100.180,434.651,174.664,21.055,153.487
C01442=1083.716,99.931,434.669,174.663,21.053,153.487
C01443=1083.710,99.682,434.687,174.660,21.050,153.486
C01444=1083.705,99.432,434.705,174.659,21.049,153.486
C01445=1083.699,99.184,434.724,174.657,21.046,153.486
C01446=1083.693,98.934,434.742,174.655,21.045,153.486
C01447=1083.688,98.685,434.760,174.653,21.042,153.486
C01448=1083.682,98.436,434.778,174.652,21.041,153.486
C01449=1083.676,98.186,434.796,174.649,21.039,153.486
C01450=1083.671,97.937,434.815,174.648,21.037,153.486
C01451=1083.665,97.688,434.833,174.645,21.035,153.486
C01452=1083.659,97.438,434.851,174.644,21.033,153.485
C01453=1083.654,97.190,434.870,174.642,21.030,153.485
C01454=1083.648,96.940,434.888,174.640,21.029,153.485
C01455=1083.642,96.691,434.905,174.638,21.027,153.485
C01456=1083.636,96.441,434.924,174.637,21.025,153.485
C01457=1083.631,96.192,434.942,174.635,21.023,153.485
C01458=1083.625,95.943,434.960,174.633,21.021,153.485
C01459=1083.619,95.664,434.981,174.631,21.018,153.485
C01460=1083.613,95.385,435.000,174.629,21.016,153.485
C01461=1083.607,95.106,435.021,174.627,21.014,153.484
C01462=1083.600,94.826,435.041,174.624,21.011,153.484
C01463=1083.593,94.577,435.059,174.623,21.010,153.484
C01464=1083.589,94.328,435.077,174.621,21.007,153.484
C01465=1083.583,94.079,435.095,174.619,21.005,153.484
C01466=1083.577,93.829,435.113,174.617,21.003,153.484
C01467=1083.572,93.580,435.130,174.616,21.001,153.484
C01468=1083.566,93.331,435.150,174.614,20.999,153.484
C01469=1083.560,93.082,435.167,174.612,20.997,153.483
C01470=1083.555,92.833,435.185,174.610,20.995,153.483
C01471=1083.549,92.583,435.203,174.608,20.993,153.483
C01472=1083.544,92.333,435.221,174.606,20.991,153.483
C01473=1083.538,92.084,435.240,174.605,20.989,153.483
C01474=1083.532,91.835,435.257,174.603,20.987,153.483
C01475=1083.526,91.586,435.275,174.601,20.985,153.483
C01476=1083.521,91.336,435.293,174.599,20.983,153.483
C01477=1083.516,91.087,435.311,174.598,20.981,153.482
C01478=1083.510,90.838,435.328,174.595,20.979,153.482
C01479=1083.504,90.588,435.346,174.594,20.977,153.482
C01480=1083.498,90.339,435.364,174.592,20.974,153.482
C01481=1083.492,90.090,435.382,174.591,20.972,153.482
C01482=1083.487,89.841,435.399,174.588,20.970,153.482
C01483=1083.480,89.591,435.418,174.587,20.969,153.482
C01484=1083.475,89.342,435.436,174.585,20.966,153.482
C01485=1083.469,89.093,435.453,174.583,20.965,153.482
C01486=1083.463,88.844,435.471,174.581,20.962,153.481
C01487=1083.458,88.595,435.489,174.580,20.960,153.481
C01488=1083.452,88.344,435.507,174.577,20.958,153.481
C01489=1083.447,88.095,435.525,174.576,20.956,153.481
C01490=1083.441,87.846,435.542,174.574,20.954,153.481
C01491=1083.435,87.597,435.560,174.572,20.952,153.481
C01492=1083.430,87.348,435.578,174.570,20.950,153.481
C01493=1083.424,87.099,435.595,174.569,20.948,153.481
C01494=1083.418,86.849,435.613,174.567,20.946,153.480
C01495=1083.412,86.600,435.631,174.565,20.944,153.480
C01496=1083.407,86.351,435.648,174.563,20.942,153.480
C01497=1083.401,86.101,435.666,174.562,20.940,153.480
C01498=1083.395,85.852,435.684,174.559,20.938,153.480
C01499=1083.390,85.602,435.701,174.558,20.936,153.480
C01500=1083.384,85.353,435.719,174.557,20.934,153.480
C01501=1083.378,85.104,435.736,174.554,20.932,153.480
C01502=1083.373,84.855,435.754,174.553,20.930,153.479
C01503=1083.367,84.605,435.772,174.551,20.927,153.479
C01504=1083.361,84.356,435.789,174.550,20.925,153.479
C01505=1083.356,84.107,435.807,174.547,20.923,153.479
C01506=1083.349,83.857,435.824,174.546,20.922,153.479
C01507=1083.343,83.608,435.842,174.544,20.919,153.479
C01508=1083.338,83.359,435.859,174.542,20.917,153.479
C01509=1083.333,83.110,435.876,174.540,20.915,153.478
C01510=1083.327,82.860,435.894,174.539,20.913,153.478
C01511=1083.321,82.611,435.912,174.536,20.911,153.478
C01512=1083.315,82.362,435.929,174.535,20.909,153.478
C01513=1083.310,82.112,435.946,174.533,20.906,153.478
C01514=1083.304,81.862,435.964,174.532,20.905,153.478
C01515=1083.299,81.613,435.982,174.529,20.902,153.478
C01516=1083.293,81.364,435.999,174.528,20.900,153.477
C01517=1083.288,81.115,436.017,174.527,20.898,153.477
C01518=1083.282,80.865,436.034,174.524,20.896,153.477
C01519=1083.276,80.616,436.052,174.523,20.894,153.477
C01520=1083.271,80.367,436.069,174.521,20.892,153.477
C01521=1083.265,80.118,436.087,174.520,20.890,153.477
C01522=1083.259,79.867,436.104,174.517,20.888,153.477
C01523=1083.253,79.589,436.123,174.515,20.885,153.476
C01524=1083.247,79.310,436.143,174.514,20.883,153.476
C01525=1083.241,79.031,436.163,174.512,20.881,153.476
C01526=1083.234,78.751,436.182,174.510,20.878,153.476
C01527=1083.228,78.502,436.199,174.508,20.876,153.476
C01528=1083.222,78.253,436.216,174.506,20.874,153.476
C01529=1083.217,78.004,436.233,174.505,20.872,153.476
C01530=1083.211,77.754,436.251,174.503,20.870,153.475
C01531=1083.206,77.505,436.268,174.501,20.868,153.475
C01532=1083.200,77.256,436.285,174.500,20.866,153.475
C01533=1083.194,77.007,436.302,174.498,20.864,153.475
C01534=1083.189,76.758,436.320,174.496,20.862,153.475
C01535=1083.182,76.508,436.337,174.494,20.859,153.475
C01536=1083.177,76.258,436.354,174.493,20.857,153.475
C01537=1083.171,76.009,436.371,174.491,20.855,153.474
C01538=1083.166,75.760,436.388,174.489,20.853,153.474
C01539=1083.160,75.511,436.405,174.487,20.851,153.474
C01540=1083.154,75.261,436.423,174.486,20.849,153.474
C01541=1083.148,75.012,436.440,174.484,20.847,153.474
C01542=1083.142,74.762,436.457,174.482,20.845,153.474
C01543=1083.137,74.513,436.474,174.481,20.843,153.474
C01544=1083.132,74.264,436.491,174.479,20.840,153.473
C01545=1083.125,74.014,436.508,174.477,20.838,153.473
C01546=1083.119,73.765,436.525,174.475,20.836,153.473
C01547=1083.114,73.515,436.543,174.474,20.834,153.473
C01548=1083.109,73.266,436.560,174.472,20.832,153.473
C01549=1083.102,73.017,436.577,174.470,20.830,153.473
C01550=1083.097,72.767,436.593,174.469,20.828,153.472
C01551=1083.092,72.518,436.611,174.467,20.825,153.472
C01552=1083.085,72.268,436.628,174.465,20.824,153.472
C01553=1083.080,72.019,436.645,174.463,20.821,153.472
C01554=1083.074,71.770,436.661,174.462,20.819,153.472
C01555=1083.068,71.521,436.679,174.460,20.817,153.472
C01556=1083.063,71.271,436.696,174.458,20.815,153.472
C01557=1083.057,71.023,436.713,174.457,20.813,153.471
C01558=1083.052,70.773,436.730,174.455,20.811,153.471
C01559=1083.046,70.523,436.746,174.454,20.809,153.471
C01560=1083.040,70.274,436.763,174.452,20.806,153.471
C01561=1083.034,70.024,436.781,174.450,20.804,153.471
C01562=1083.028,69.775,436.798,174.448,20.802,153.471
C01563=1083.023,69.526,436.814,174.447,20.800,153.471
C01564=1083.017,69.276,436.831,174.445,20.798,153.470
C01565=1083.011,69.027,436.848,174.443,20.795,153.470
C01566=1083.006,68.778,436.865,174.442,20.793,153.470
C01567=1083.000,68.528,436.881,174.440,20.791,153.470
C01568=1082.995,68.279,436.899,174.438,20.790,153.470
C01569=1082.989,68.030,436.915,174.437,20.788,153.470
C01570=1082.983,67.780,436.932,174.435,20.785,153.470
C01571=1082.977,67.531,436.949,174.433,20.783,153.469
C01572=1082.971,67.281,436.966,174.431,20.781,153.469
C01573=1082.965,67.032,436.983,174.430,20.779,153.469
C01574=1082.960,66.783,437.000,174.428,20.776,153.469
C01575=1082.954,66.533,437.016,174.427,20.774,153.469
C01576=1082.949,66.284,437.033,174.425,20.772,153.469
C01577=1082.943,66.034,437.049,174.423,20.770,153.468
C01578=1082.937,65.786,437.066,174.422,20.768,153.468
C01579=1082.931,65.536,437.083,174.420,20.766,153.468
C01580=1082.925,65.287,437.100,174.418,20.764,153.468
C01581=1082.920,65.037,437.116,174.417,20.762,153.468
C01582=1082.914,64.788,437.133,174.415,20.759,153.468
C01583=1082.909,64.539,437.150,174.413,20.757,153.467
C01584=1082.903,64.289,437.166,174.411,20.755,153.467
C01585=1082.897,64.040,437.183,174.410,20.753,153.467
C01586=1082.891,63.790,437.200,174.409,20.751,153.467
C01587=1082.884,63.511,437.219,174.407,20.748,153.467
C01588=1082.878,63.233,437.237,174.404,20.746,153.467
C01589=1082.871,62.953,437.256,174.402,20.744,153.467
C01590=1082.865,62.674,437.274,174.401,20.742,153.466
C01591=1082.859,62.425,437.290,174.399,20.739,153.466
C01592=1082.853,62.175,437.307,174.397,20.737,153.466
C01593=1082.848,61.926,437.323,174.396,20.735,153.466
C01594=1082.842,61.676,437.340,174.394,20.733,153.466
C01595=1082.835,61.427,437.357,174.393,20.731,153.466
C01596=1082.829,61.177,437.373,174.391,20.728,153.465
C01597=1082.824,60.928,437.390,174.389,20.726,153.465
C01598=1082.818,60.678,437.406,174.388,20.724,153.465
C01599=1082.812,60.429,437.423,174.386,20.722,153.465
C01600=1082.806,60.180,437.439,174.384,20.720,153.465
C01601=1082.800,59.930,437.455,174.382,20.718,153.465
C01602=1082.795,59.681,437.472,174.381,20.716,153.465
C01603=1082.789,59.431,437.488,174.379,20.714,153.464
C01604=1082.783,59.182,437.505,174.377,20.712,153.464
C01605=1082.777,58.933,437.521,174.376,20.710,153.464
C01606=1082.772,58.683,437.538,174.375,20.708,153.464
C01607=1082.766,58.434,437.554,174.373,20.705,153.464
C01608=1082.760,58.184,437.570,174.371,20.703,153.464
C01609=1082.754,57.935,437.586,174.369,20.701,153.463
C01610=1082.748,57.686,437.603,174.368,20.699,153.463
C01611=1082.743,57.436,437.620,174.366,20.697,153.463
C01612=1082.737,57.187,437.636,174.364,20.695,153.463
C01613=1082.731,56.937,437.652,174.363,20.693,153.463
C01614=1082.725,56.689,437.668,174.361,20.690,153.463
C01615=1082.719,56.439,437.684,174.360,20.688,153.462
C01616=1082.713,56.190,437.700,174.358,20.686,153.462
C01617=1082.708,55.940,437.717,174.356,20.684,153.462
C01618=1082.702,55.691,437.734,174.355,20.682,153.462
C01619=1082.696,55.442,437.750,174.353,20.680,153.462
C01620=1082.690,55.192,437.766,174.351,20.677,153.462
C01621=1082.684,54.943,437.782,174.350,20.675,153.461
C01622=1082.679,54.693,437.798,174.348,20.673,153.461
C01623=1082.674,54.443,437.815,174.347,20.671,153.461
C01624=1082.668,54.194,437.831,174.345,20.669,153.461
C01625=1082.662,53.944,437.847,174.343,20.666,153.461
C01626=1082.656,53.695,437.863,174.342,20.664,153.461
C01627=1082.650,53.446,437.879,174.341,20.662,153.460
C01628=1082.644,53.197,437.896,174.339,20.660,153.460
C01629=1082.639,52.947,437.911,174.337,20.658,153.460
C01630=1082.633,52.698,437.927,174.335,20.655,153.460
C01631=1082.628,52.448,437.944,174.334,20.653,153.460
C01632=1082.622,52.199,437.961,174.332,20.651,153.460
C01633=1082.616,51.949,437.977,174.330,20.649,153.459
C01634=1082.610,51.700,437.993,174.329,20.647,153.459
C01635=1082.605,51.451,438.008,174.328,20.645,153.459
C01636=1082.599,51.202,438.024,174.326,20.642,153.459
C01637=1082.593,50.952,438.041,174.324,20.640,153.459
C01638=1082.587,50.703,438.057,174.322,20.638,153.459
C01639=1082.581,50.453,438.073,174.321,20.636,153.458
C01640=1082.576,50.203,438.089,174.320,20.634,153.458
C01641=1082.571,49.955,438.105,174.318,20.631,153.458
C01642=1082.565,49.705,438.122,174.316,20.629,153.458
C01643=1082.559,49.455,438.137,174.315,20.627,153.458
C01644=1082.553,49.206,438.153,174.313,20.625,153.458
C01645=1082.547,48.957,438.170,174.312,20.622,153.457
C01646=1082.542,48.707,438.185,174.310,20.620,153.457
C01647=1082.536,48.458,438.201,174.308,20.618,153.457
C01648=1082.530,48.209,438.217,174.307,20.616,153.457
C01649=1082.525,47.959,438.233,174.305,20.614,153.457
C01650=1082.519,47.709,438.249,174.304,20.612,153.456
C01651=1082.513,47.429,438.267,174.302,20.609,153.456
C01652=1082.507,47.151,438.285,174.300,20.607,153.456
C01653=1082.500,46.871,438.303,174.298,20.604,153.456
C01654=1082.494,46.592,438.321,174.297,20.602,153.456
C01655=1082.488,46.342,438.336,174.295,20.599,153.455
C01656=1082.482,46.093,438.352,174.294,20.597,153.455
C01657=1082.476,45.844,438.369,174.291,20.595,153.455
C01658=1082.471,45.594,438.384,174.290,20.592,153.455
C01659=1082.465,45.345,438.400,174.289,20.590,153.455
C01660=1082.460,45.095,438.416,174.287,20.588,153.454
C01661=1082.454,44.846,438.432,174.286,20.586,153.454
C01662=1082.449,44.596,438.447,174.284,20.584,153.454
C01663=1082.443,44.347,438.463,174.282,20.581,153.454
C01664=1082.437,44.098,438.480,174.281,20.579,153.454
C01665=1082.432,43.849,438.495,174.280,20.577,153.454
C01666=1082.426,43.599,438.511,174.278,20.575,153.453
C01667=1082.420,43.349,438.527,174.276,20.573,153.453
C01668=1082.414,43.100,438.543,174.275,20.571,153.453
C01669=1082.409,42.850,438.558,174.273,20.568,153.453
C01670=1082.403,42.601,438.574,174.272,20.566,153.453
C01671=1082.397,42.352,438.589,174.270,20.564,153.453
C01672=1082.391,42.102,438.605,174.268,20.561,153.452
C01673=1082.385,41.852,438.621,174.267,20.559,153.452
C01674=1082.380,41.604,438.637,174.266,20.557,153.452
C01675=1082.374,41.354,438.652,174.264,20.555,153.452
C01676=1082.369,41.104,438.668,174.262,20.553,153.452
C01677=1082.363,40.855,438.683,174.261,20.551,153.451
C01678=1082.357,40.605,438.699,174.259,20.548,153.451
C01679=1082.351,40.356,438.715,174.258,20.546,153.451
C01680=1082.345,40.106,438.731,174.257,20.544,153.451
C01681=1082.340,39.857,438.747,174.254,20.542,153.451
C01682=1082.334,39.608,438.761,174.253,20.540,153.451
C01683=1082.328,39.358,438.777,174.252,20.538,153.450
C01684=1082.323,39.109,438.793,174.250,20.535,153.450
C01685=1082.317,38.859,438.808,174.248,20.533,153.450
C01686=1082.311,38.610,438.825,174.247,20.531,153.450
C01687=1082.305,38.361,438.839,174.245,20.528,153.450
C01688=1082.300,38.111,438.855,174.244,20.526,153.449
C01689=1082.294,37.862,438.871,174.243,20.524,153.449
C01690=1082.289,37.612,438.886,174.240,20.522,153.449
C01691=1082.282,37.363,438.901,174.239,20.520,153.449
C01692=1082.276,37.113,438.917,174.238,20.518,153.449
C01693=1082.271,36.863,438.933,174.236,20.515,153.449
C01694=1082.265,36.614,438.948,174.234,20.513,153.448
C01695=1082.259,36.364,438.963,174.233,20.511,153.448
C01696=1082.252,36.115,438.979,174.231,20.508,153.448
C01697=1082.247,35.866,438.994,174.230,20.506,153.448
C01698=1082.242,35.616,439.009,174.229,20.504,153.448
C01699=1082.235,35.367,439.025,174.226,20.502,153.448
C01700=1082.230,35.118,439.040,174.225,20.500,153.447
C01701=1082.224,34.868,439.056,174.224,20.498,153.447
C01702=1082.218,34.618,439.071,174.222,20.496,153.447
C01703=1082.213,34.370,439.087,174.220,20.494,153.447
C01704=1082.206,34.120,439.102,174.219,20.491,153.447
C01705=1082.201,33.870,439.117,174.217,20.489,153.446
C01706=1082.196,33.621,439.132,174.216,20.487,153.446
C01707=1082.189,33.371,439.147,174.215,20.485,153.446
C01708=1082.183,33.122,439.164,174.212,20.482,153.446
C01709=1082.177,32.873,439.178,174.211,20.480,153.446
C01710=1082.172,32.623,439.194,174.210,20.478,153.446
C01711=1082.167,32.373,439.209,174.208,20.475,153.445
C01712=1082.160,32.124,439.224,174.207,20.473,153.445
C01713=1082.154,31.874,439.240,174.205,20.471,153.445
C01714=1082.149,31.625,439.255,174.204,20.469,153.445
C01715=1082.142,31.346,439.272,174.202,20.467,153.445
C01716=1082.136,31.066,439.288,174.200,20.464,153.444
C01717=1082.130,30.787,439.306,174.199,20.462,153.444
C01718=1082.123,30.507,439.323,174.197,20.459,153.444
C01719=1082.117,30.258,439.338,174.195,20.457,153.444
C01720=1082.112,30.008,439.353,174.194,20.455,153.444
C01721=1082.105,29.759,439.369,174.192,20.453,153.443
C01722=1082.100,29.510,439.384,174.191,20.451,153.443
C01723=1082.094,29.260,439.399,174.190,20.448,153.443
C01724=1082.088,29.010,439.414,174.188,20.446,153.443
C01725=1082.082,28.762,439.429,174.186,20.444,153.443
C01726=1082.077,28.512,439.444,174.185,20.442,153.442
C01727=1082.071,28.263,439.459,174.183,20.439,153.442
C01728=1082.065,28.013,439.475,174.182,20.437,153.442
C01729=1082.060,27.764,439.489,174.180,20.435,153.442
C01730=1082.054,27.514,439.505,174.178,20.433,153.442
C01731=1082.048,27.264,439.520,174.177,20.430,153.442
C01732=1082.042,27.015,439.534,174.176,20.428,153.441
C01733=1082.036,26.765,439.550,174.174,20.426,153.441
C01734=1082.030,26.516,439.564,174.172,20.424,153.441
C01735=1082.025,26.266,439.580,174.171,20.422,153.441
C01736=1082.019,26.017,439.595,174.170,20.420,153.441
C01737=1082.013,25.768,439.609,174.168,20.417,153.441
C01738=1082.007,25.518,439.625,174.167,20.415,153.440
C01739=1082.001,25.269,439.640,174.165,20.413,153.440
C01740=1081.995,25.019,439.655,174.164,20.411,153.440
C01741=1081.990,24.770,439.670,174.162,20.408,153.440
C01742=1081.983,24.520,439.685,174.161,20.406,153.440
C01743=1081.978,24.271,439.700,174.159,20.405,153.439
C01744=1081.972,24.021,439.714,174.157,20.402,153.439
C01745=1081.966,23.772,439.729,174.156,20.400,153.439
C01746=1081.961,23.522,439.744,174.155,20.398,153.439
C01747=1081.955,23.273,439.759,174.153,20.395,153.439
C01748=1081.949,23.023,439.774,174.151,20.393,153.439
C01749=1081.944,22.774,439.789,174.150,20.391,153.438
C01750=1081.937,22.524,439.804,174.149,20.389,153.438
C01751=1081.931,22.275,439.818,174.147,20.387,153.438
C01752=1081.926,22.025,439.833,174.146,20.384,153.438
C01753=1081.920,21.776,439.848,174.144,20.382,153.438
C01754=1081.914,21.526,439.863,174.142,20.380,153.437
C01755=1081.909,21.277,439.878,174.141,20.378,153.437
C01756=1081.902,21.027,439.893,174.140,20.376,153.437
C01757=1081.897,20.778,439.907,174.138,20.374,153.437
C01758=1081.891,20.528,439.922,174.136,20.371,153.437
C01759=1081.886,20.279,439.937,174.135,20.369,153.436
C01760=1081.879,20.029,439.952,174.134,20.367,153.436
C01761=1081.873,19.780,439.966,174.132,20.364,153.436
C01762=1081.868,19.531,439.981,174.130,20.362,153.436
C01763=1081.862,19.280,439.996,174.129,20.360,153.436
C01764=1081.856,19.031,440.010,174.128,20.358,153.436
C01765=1081.850,18.782,440.025,174.126,20.356,153.436
C01766=1081.844,18.533,440.040,174.125,20.353,153.435
C01767=1081.838,18.283,440.054,174.123,20.351,153.435
C01768=1081.833,18.033,440.069,174.122,20.349,153.435
C01769=1081.827,17.784,440.084,174.120,20.347,153.435
C01770=1081.821,17.534,440.098,174.119,20.345,153.435
C01771=1081.815,17.284,440.113,174.117,20.343,153.434
C01772=1081.809,17.035,440.128,174.115,20.341,153.434
C01773=1081.804,16.786,440.143,174.114,20.338,153.434
C01774=1081.798,16.536,440.157,174.113,20.336,153.434
C01775=1081.792,16.287,440.172,174.112,20.334,153.434
C01776=1081.786,16.037,440.187,174.109,20.332,153.433
C01777=1081.780,15.788,440.200,174.108,20.330,153.433
C01778=1081.774,15.538,440.215,174.107,20.328,153.433
C01779=1081.768,15.239,440.232,174.105,20.325,153.433
C01780=1081.761,14.939,440.250,174.103,20.322,153.433
C01781=1081.754,14.639,440.268,174.102,20.320,153.432
C01782=1081.747,14.339,440.285,174.100,20.317,153.432
C01783=1081.741,14.090,440.300,174.099,20.315,153.432
C01784=1081.735,13.841,440.315,174.096,20.312,153.432
C01785=1081.729,13.591,440.328,174.095,20.310,153.432
C01786=1081.723,13.341,440.343,174.094,20.308,153.431
C01787=1081.717,13.092,440.357,174.093,20.306,153.431
C01788=1081.712,12.843,440.372,174.090,20.304,153.431
C01789=1081.706,12.593,440.386,174.089,20.302,153.431
C01790=1081.700,12.344,440.401,174.088,20.300,153.431
C01791=1081.693,12.094,440.416,174.087,20.298,153.431
C01792=1081.688,11.844,440.430,174.084,20.295,153.431
C01793=1081.682,11.595,440.444,174.083,20.293,153.430
C01794=1081.676,11.345,440.458,174.082,20.291,153.430
C01795=1081.670,11.096,440.473,174.080,20.288,153.430
C01796=1081.664,10.846,440.487,174.079,20.286,153.430
C01797=1081.658,10.597,440.501,174.077,20.284,153.430
C01798=1081.652,10.348,440.515,174.076,20.282,153.429
C01799=1081.646,10.098,440.530,174.074,20.280,153.429
C01800=1081.640,9.849,440.544,174.073,20.278,153.429
C01801=1081.634,9.599,440.559,174.071,20.276,153.429
C01802=1081.629,9.349,440.573,174.070,20.274,153.429
C01803=1081.623,9.100,440.586,174.068,20.271,153.429
C01804=1081.617,8.850,440.601,174.067,20.269,153.428
C01805=1081.611,8.600,440.615,174.066,20.267,153.428
C01806=1081.605,8.352,440.630,174.064,20.265,153.428
C01807=1081.599,8.101,440.644,174.062,20.262,153.428
C01808=1081.594,7.852,440.659,174.061,20.260,153.428
C01809=1081.588,7.603,440.673,174.060,20.258,153.427
C01810=1081.582,7.352,440.687,174.058,20.257,153.427
C01811=1081.576,7.103,440.701,174.056,20.254,153.427
C01812=1081.570,6.854,440.715,174.055,20.252,153.427
C01813=1081.564,6.605,440.730,174.054,20.250,153.427
C01814=1081.558,6.355,440.743,174.053,20.248,153.427
C01815=1081.553,6.105,440.757,174.051,20.245,153.426
C01816=1081.546,5.856,440.772,174.049,20.243,153.426
